(* Version history:
Date	|	Version/Author |	Remark
----------------------------------------------------------------------------------------------------
11.09.01	|	2.01 JP		|	new version depending on 0.99D
22.11.01	|	2.02 JP		|	new version depending on 0.99F
18.01.02	|	2.03 JP		|	new version depending on 1.0
		|				|	changed names, interfaces, execute behavior
25.01.02	|	2.04 JP		|	no CAMMING, change behavior of MC_Power
07.02.02	|	2.05 JP		|	SetOverride in unit less than 1%
13.02.02	|	2.06 JP		|	New: MC_NewPos and MC_NewPosAndVelo
		|				|	removed MC_MoveAdditive
14.02.02	|	2.07 JP		|	completed: MC_Home, MC_MoveSuperImposed
14.02.02	|	2.08 JP		|	renamed MC_NewPosAndVelo New: MC_SetOverride edge triggered
15.02.02	|	2.09 JP		|	changed: MC_Gear
15.02.02	|	2.10 JP		|	changed: MC_SetOverride
04.04.02	|	2.11 JP		|	changed: done for MC_Home 
		|				|	new: Check TimeOut for MoveAbsolute, MoveRelative, Home
08.03.02	|	2.12 JP		|	changed: new flag inserted 
12.03.02	|	2.13 JP		|	changed: reset of bNotExecute
18.03.02	|	2.14 JP		|	changed: MC_Reset waits for ready
22.03.02	|	2.15 JP		|	changed: MC_Read and Write FBs
26.03.02	|	2.16 JP		|	revised: Read/Write Parameter FBs
27.03.02	|	2.17 JP		|	revised: Read/Write Parameter FBs and Home (calibration cam)
09.04.02	|	2.18 JP		|	changed parameter type of some parameters
17.04.02	|	2.19 JP		|	changed: Read(Bool)Parameter new Input to select read mode
							Boolean parameters can be read with ReadParameter
							changed MC_Power: new input override !!			
23.04.02	|	2.20 JP		|	fixed: MC_Home changed: Behavior of MC_MoveAbsolute/Relative
25.04.02	|	2.21 JP		|	changed: MC_Reset: now not waiting for 'axis is ready'. Check with MC_Power !
26.04.02	|	2.22 JP		|	MC_Home: If Posistion =  DEFAULT_HOME_POSITION --> no set of position
							MC_MoveXX: more detailed error messages
05.07.02	|	2.23 JP		|	new MC_MoveAbsoluteOrRestart: combines MoveAbsolute and NewPos
19.07.02	|	2.24 JP		|	changed: E_STATES ---> E_TCMC_STATES
12.09.02	|	2.25 KST		|	changed: MC_MoveAbsolute and MC_MoveRelative now based on FB_MoveGeneric
							MC_NewPos and MC_NewPosAndVelo based on new FB_NewPosAndVeloGeneric 
							new internal start types in MC_MoveAbsoluteOrRestart (message suppression)
16.09.02	|	2.26 ChristophC|	changed: MC_SetActualPosition due to changes in TcNC.Lib
16.10.02	|	2.27 KST		|	new: MC_ExtSetPointGenEnable and MC_ExtSetPointGenDisable
29.10.02	|	2.28 ChristophC|	MC_Stop and MC_SetActualPosition: Ads port changed from TcMcGlobal.NCPORT_TCMC => AMSPORT_R0_NCSAF
12.11.02	|	2.29 ChristophC|	MC_OverrideFilter function block added
13.12.02	|	2.30 JP		|	several smaller changes: MC_ReadStatus, MC_Stop
22.01.03	|	2.31 KSt		|	new additional function MC_ExtSetPointGenFeed
24.03.03	|	2.32 JP		|	added: MC_GearFloat, corr. MC_ReadBoolParameter (wrong for AxisEnPostionRangeMonitoring)
26.03.03	|	2.33 KSt		|	added: MC_MoveModulo
04.04.03	|	2.34 KSt		|	changed: MC_MoveAbsoluteOrRestart, Done will be reset at once after Execute=FALSE
12.05.03	|	2.35 JP		|	changed: MC_MoveVelocity, MC_Home (error handling), MC_ReadStatus
14.05.03	|	2.36 KSt		|	changed: MC_Home, MC_MoveAbsoluteOrRestart
15.05.03	|	2.36.1 KSt	|	changed: MC_Home
28.05.03	|	2.37 KSt		|	changed: MC_MoveVelocity, abort during acceleration phase	
							changed: MC_MoveAbsoluteOrRestart, reset internal error on restart
27.06.03	|	2.38 JP		|	changed: MC_Stop: Execute behavior
22.07.03	|	2.38.1 KSt	|	added: new error codes
12.08.03	|	2.39 KSt		|	changed: FB_ReadWriteParameter, size of bool parameters
15.08.03	|	2.40 KSt		|	added: new block MC_ChangeDynParam
19.08.03	|	2.41 JP		|	changed: MC_ReadParameter: Done falls with Execute
01.10.03	|	2.42 KSt		|	changed: MC_MoveAbsoluteOrRestart, Execute directly after done issue fixed
09.10.03	|	2.43 KSt		|	new function block MC_SetReferenceFlag
04.12.03	|	2.44 KSt		|	ReadBoolParameter(AxisEnTargetPositionMonitoring) corrected
12.01.04	|	2.45 KSt		|	MC_MoveSuperimposed revised
						|	R_Trigger(execute) moved outside CASE in all move function blocks
19.01.04	|	2.45.1 KSt	|	Busy Signal in MC_MoveSuperimposed
30.04.04	|	2.46.0 KSt	|	New function blocks MC_TouchProbe, MC_AbortTrigger, internal block MC_OrientedStop
						|	MC_ReadParameter revised
06.05.04	|	2.46.1 KSt	|	Correction in MC_OrientedStop
21.05.04	|	2.47.0 KSt	|	MC_GearInDyn added - master slave coupling with dynamic gear ratio
06.08.04	|	2.47.1 KSt	|	MC_OrientedStop moved from internal to additional folder
						|	MC_MoveAbsoluteOrRestart additional internal error code NC_ERROR_STARTINTERNAL_NOTREADY evaluated
23.08.04	|	2.47.2 KSt	|	new local flag EmergencyStop in MC_Stop signals type of internal ADS stop command
10.01.05	|	2.47.3 KSt	|	new function block MC_MoveSuperImposedExt
28.01.05	|	2.47.4 KSt	|	TcMcGlobal.tTargetPosTimeOut changed from 5 sec to 6 sec to be later than a NC PEH error (5 sec)
15.02.05	|	2.48.0 KSt	|	new function block MC_GearOutExt 
28.02.05	|	2.49.0 JP		|	Execute and Done behavior corrected for MC_ReadActualPos and MC_SetActualPos
10.03.05	|	2.50.0 KSt	|	all function blocks use a global AMS net-ID TcMcGlobal.NCNETID_TCMC which may be modified by the user
17.03.05	|	2.51.0 KSt	|	new function block MC_PowerStepper
						|	MC_MoveAbsoluteOrRestart restart while starting (adswrite.Busy) changed
24.05.05	|	2.52.0 KSt	|	acceleration added to block MC_GearOutExt 
05.07.05	|	2.53.0 KSt	|	new local flag ADSbusy in all function blocks
05.07.05	|	2.54.0 KSt	|	new function block MC_GearInDynCCV
06.07.05	|	2.55.0 KSt	|	Busy timing improved in all function blocks (turns immediately to FALSE with Done or Error or Aborted)
25.07.05	|	2.55.1 KSt	|	Change for status output behavior 
26.07.05	|	2.55.2 KSt	|	MC_GearOutExt extended through mode 'oriented stop'
03.08.05	|	2.55.3 KSt	|	Commands MC_MoveAbsoluteOrRestart, MC_NewPos and MC_NewPosAndVelo now directed to port AMSPORT_R0_NCSAF
						|	Summary of other commands to SAF: MC_Stop, MC_OrientedStop, MC_TouchProbe, MC_AbortTrigger, MC_SetReferenceFlag, MC_PowerStepper
14.09.05	|	2.56.0 KSt	|	new function block MC_ParameterizedStop
26.09.05	|	2.56.1 KSt	|	Jerk parameter added to MC_ChangeDynParam. Block moved into the internal folder.
07.11.05	|	2.56.2 KSt	|	internal block FB_ReadCharacteristicValues changed to ADSRDWRT
19.12.05	|	2.56.3 KSt	|	new block MC_SetActualPositionOnTheFly
05.01.06	|	2.56.4 KSt	|	new blocks MC_ReadParameterSet and MC_ReadAxisComponents
21.02.06	|	2.57.0 KSt	|	NC status feedback monitoring changed in MC_GearIn and MC_GearInFloat
29.03.06	|	2.57.1 KSt	|	new order of the blocks in the library tree
11.04.06	|	2.57.2 HKP	|	Command MC_ChangeDynParam now directed to port AMSPORT_R0_NCSAF
10.05.06	|	2.57.3 KSt	|	new function block MC_Jog
17.05.06	|	2.57.4 KSt	|	MC_Jog: MC_JOGMODE_INCHING_MODULO temporarily deactivated
05.07.06	|	2.57.5 KSt	|	NC status feedback monitoring changed in MC_GearInDyn and MC_GearInDynCCV
=======	|===============	|==========================================================================
12.07.06	|	2.57.6 KSt	|	new AMS port NCPORT_TCMC_COUPLING for all coupling commands
11.08.06	|	2.57.7 KSt	|	reset Done when Execute is FALSE in FB_NewPosAndVeloGeneric
						|	MC_Jog released
22.08.06	|	2.57.8 KSt	|	new function block MC_AbortSuperposition
07.11.06	|	2.57.9 HKP	|	changes in function block MC_PowerStepper
06.02.07	|	2.57.10 KSt	|	initialization problem with modulo positions fixed in MC_TouchProbe.
						|	recorded position at PlcEvent now modulo when requested.
14.03.07	|	2.57.11 KSt	|	MC_Jog: Handling of CommandAborted corrected
24.04.07	|	2.57.12 KSt	|	additional parameters in MC_AxisPara, MC_ReadParameters, MC_WriteParameters
31.05.07	|	2.57.13 KSt	|	FPU exception with LREAL_TO_BOOL and DWORD_TO_BOOL fixed in FB_ReadWriteParameter 
12.06.07	|	2.57.14 KSt	|	FB_NewPosAndVeloGeneric and MC_MoveSuperImposed(Ext): IF condition changed from "NOT AxisIsMoving" to "NOT AxisHasJob"
=======	|===============	|==========================================================================
12.06.07	|	2.57.14 KSt	|	TcMC2 development started - following 2.xx.xx changes have been added in parallel
02.11.07	|	2.57.15 KSt	|	data structure ST_TableCharacValues extended
18.12.07	|	2.57.16 KSt	|	MC_Jog is now internally using MC_MoveRelative instead of MC_MoveAbsolute to work with backlash compensation
20.05.08	|	2.57.18 KSt	|	AxisModuloPositionFlag added to MC_ReadBoolParameter
17.06.08	|	2.57.20 KSt	|	MC_GearInMultiMaster added
24.07.08	|	2.57.22 KSt	|	MC_Power supports now a minimum Enable-Off/On toggle time of 50ms to reenable the Status output
28.10.08	|	2.57.23 KSt	|	new function block MC_SetEncoderScalingFactor
=======	|===============	|==========================================================================
16.03.07	|	3.00.00 KSt	|	new version depending on PLCopen V1.1 (beta)
25.08.08   |	3.00.01 KSt	|	released as TcMC2 
17.09.08   |	3.00.02 KSt	|	last result added in MC_Reset
26.11.08   |	3.00.03 KSt	|	change in MC_Stop and MoveGeneric for delayed error handling
01.12.08   |	3.00.04 KSt	|	MC_Stop - Done is set immediately at standstill
18.12.08   |	3.00.05 KSt	|	MC_Power - uses now ControlLoopClosed instead of AxisIsReady
13.01.09   |	3.00.06 KSt	|	independent characteristic data for camming and flying saw
16.01.09   |	3.00.07 KSt	|	all move commands: changed handling of CmdNo=0 and CmdNo+2 leads to better results (CommandAborted)
23.01.09   |	3.00.08 KSt	|	MC_MoveSuperimposed is now passed to port AMSPORT_R0_NCSAF (501)
28.01.09   |	3.00.09 KSt	|	Homing mode MC_Direct added - Mode option for MC_SetPosition added
29.01.09   |	3.00.10 KSt	|	Warning output added to MC_MoveSuperimposed
05.02.09   |	3.00.11 KSt	|	axis state is now DISABLED if control loop is not closed (was STANDSTILL for virtual axes - _F_AxisState)
05.02.09   |	3.00.11 KSt	|	all move commands: CmdNo=0 is ignored as invalid - change of the coupled state leads to CommandAborted
06.02.09   |	3.00.11 KSt	|	errors on missing cyclic NC command feedback are delayed for a few cycles to avoid problems with multiple function block calls during one PLC cycle
19.02.09   |	3.00.12 KSt	|	MC_GearInDyn and MC_GearInMultimaster - no reset of gear ratio after Enable is reset to FALSE
24.02.09   |	3.01.00 KSt	|	Motion commands on slaves (must be enabled in the axis parameters before)
12.03.09   |	3.01.01 KSt	|	MC_Jog - Active output added - reset outputs when Execute is false 
09.04.09   |	3.01.02 KSt	|	MC_SetPosition and MC_SetEncoderScalingFactor - explicit encoder / control loop index 0..n can be selected
15.04.09   |	3.01.03 KSt	|	MC_Stop - outputs (except Busy) are reset after Execute=FALSE - can be retriggered during release phase
17.04.09   |	3.01.04 KSt	|	MC_Home - static homing with DEFAULT_HOME_POSITION implemented - Option.ClearPositionLag available 
11.05.09   |	3.01.05 KSt	|	MC_Stop - incorrect error message 4B63 removed;  
30.06.09   |	3.01.06 KSt	|	MC_MoveSuperimposed - new types ACCREDUCTION - new AbortOptions
28.07.09   |	3.01.07 KSt	|	MC_ExtSetPointGenFeed feeds additional counter information to the NC
13.08.09   |	3.01.08 KSt	|	MC_MoveSuperimposed - new AbortOptions - Done behavior adapted
01.09.09   |	3.01.09 KSt	|	MC_SetPosition - new option 'set absolute measuring'
30.09.09   |	3.01.10 KSt	|	MC_MoveSuperimposed - fix for new AbortOptions - HasJob flag not required before starting the command
06.10.09   |	3.01.11 KSt	|	MC_Stop - wait extra cycles before axis release error 
06.10.09   |	3.01.12 KSt	|	MC_MoveSuperimposed - fix for new AbortOptions - HasJob or IsMoving check at beginning and end of compensation 
07.10.09   |	3.01.13 KSt	|	MC_MoveSuperimposed - initial motion check removed for new AbortOptions
28.10.09   |	3.01.14 KSt	|	MC_ExtSetPointGenEnable/Disable - port changed from SVB to SAF
06.11.09   |	3.01.15 KSt	|	MC_SetPosition - new option 'set absolute measuring' removed
09.11.09   |	3.01.16 KSt	|	MC_Stop on slave axes was not rejected with error - fixed
18.11.09   |	3.01.17 KSt	|	MC_Jog - usage with protected (coupled) axes refused
26.11.09   |	3.01.18 KSt	|	Axis status data: UpdateCycleTime calculation fixed
08.12.09   |	3.01.19 KSt	|	_FB_MoveGeneric - mapping check to avoid early Error and CommandAborted signals
25.02.10   |	3.01.20 KSt	|	MC_MoveSuperimposed - additional outputs ActualAcceleration and ActualDeceleration
11.03.10   |	3.01.21 KSt	|	MC_Power - no Enable timeout error for coupled axes
07.04.10   |	3.01.22 KSt	|	MC_ReadApplicationRequest added
15.04.10   |	3.01.23 KSt	|	MC_PositionCorrectionLimiter added - cyclic update of UpdateTaskIndex and UpdateCycleTime removed from ReadStatus
23.04.10   |	3.01.24 KSt	|	internal MC_TouchProbe_V2_00 for new multi probe interface
04.05.10   |	3.01.25 KSt	|	fix in MC_WriteParameter to write bool parameters with MC_WriteParameter as well as MC_WriteBoolParameters
06.05.10   |	3.01.25 KSt	|	fix in MC_MoveContinous... for output InEndVelocity
31.05.10   |	3.02.00 KSt	|	_TcMC_ADS commands added to allow PLC running faster than NC, added to MC_Reset
08.07.10   |	3.02.01 KSt	|	fix in NC mapping counter monitoring (time-out check)
24.09.10   |	3.02.02 KSt	|	ST_NcApplicationRequest structure extended
27.10.10   |	3.02.03 KSt	|	MC_TouchProbe - TRUNC function replaced by MODABS for modulo calculations
22.11.10	|	3.02.04 KSt	|	MC_Power - axis will be enabled automatically after Error turns to FALSE and control loop is closed (just if Enable=TRUE)
		|				|	Move-Commands on axes with external set point generator (must be enabled in the axis parameters before)
29.11.10	|	3.02.05 KSt	|	MC_ReadParameter - new parameters AxisCycleTime NcSafCycleTime and NcSvbCycleTime
17.01.11	|	3.02.06 KSt	|	Phasing blocks added
21.01.11	|	3.02.06 KSt	|	MC_ExtSetPointGenEnable and MC_ExtSetPointGenDisable: code rewritten in ST
16.02.11	|	3.02.07 KSt	|	MC_TouchProbe and MC_TouchProbe_V2_00 - correction for WindowOnly with FirstPosition>LastPosition
18.02.11	|	3.02.08 KSt	|	MC_TouchProbe_V2_00 - TRIGGER_REF extended by optional physical input definition 
21.02.11	|	3.02.08 KSt	|	_MC_Phasing beta version included
25.03.11	|	3.02.09 KSt	|	minor adaption to PlcOpen V2.0 "Function blocks for motion control" released document.
05.04.11	|	3.02.10 KSt	|	new parameters defined for fast axis stopp 
21.04.11	|	3.02.11 KSt	|	FB_MoveUniversalGeneric - fix in command number overrun calculation 
27.04.11	|	3.02.12 KSt	|	new function block MC_ReadStopInfo to read the expected distance and time to stop an axis
02.05.11	|	3.02.13 KSt	|	dynamical data for fast axis stopp can be read or written by MC_ReadParameter, MC_WriteParameter
03.05.11	|	3.02.14 KSt	|	MC_TouchProbe_V2_00 - additional output data structure MC_TouchProbeRecordedData 
11.05.11	|	3.02.15 KSt	|	type check adaptions for the PLC3 compiler
18.05.11	|	3.02.16 KSt	|	data types ST_AxisParameterSet and ST_NcApplicationRequest extended
31.05.11	|	3.02.17 HKP	|	Check of AxisIsReady removed from MC_MoveCommands
31.05.11	|	3.02.17 KSt	|	Axis.OpMode.SimulationAxis added
29.06.11	|	3.02.18 KSt	|	MC_ReadParameterSet fixed for use with differently aligned systems (ARM)
12.07.11	|	3.02.19 KSt	|	internal storage added to AXIS_REF
19.07.11	|	3.02.20 KSt	|	Two Speed Axes: InVelocity detection fixed in MC_MoveVelocity
01.08.11	|	3.02.21 KSt	|	Check of cyclic motion command call - 'buffered command monitoring error' changed to 'cyclic call error' if not cyclically called
07.09.11	|	3.02.22 KSt	|	optional advanced slave motion profile for MC_GearInMultiMaster
13.10.11	|	3.02.23 KSt	|	new OpMode flag AllowExtSetAxisCommands
08.12.11	|	3.02.25 KSt	|	stop monitoring for stop and halt commands added (comparable with target position monitoring)
22.12.11	|	3.02.26 KSt	|	MC_Reset fixed for short PLC cycle times (_TcMC_ADSWRITE waits 2 cycles for NC process image)
22.12.11	|	3.02.27 KSt	|	MC_GearOut and MC_CamOut are now waiting for the NC couple state feedback in Nc2Plc
19.01.12	|	3.02.28 KSt	|	MC_TouchProbe_V2 released
23.02.12	|	3.02.29 ICh	|	_ST_TcNc_OperationModes: cleanup, StopMonitoring added, _ST_TcNC_SetPos: fReserved added to match NC definition
23.02.12	|	3.02.30 KSt	|	typecasts for TC3 to avoid TC3 compiler messages
23.03.12	|	3.02.31 KSt	|	initialization code for MoveModulo revised 
16.05.12	|	3.02.32 KSt	|	MC_MoveVelocity: InVelocity is now reset after abortion or error
05.07.12	|	3.02.33 KSt	|	state diagram changed - if axis has error, state is always ERRORSTOP (never DISABLED)
27.07.12	|	3.02.34 KSt	|	new function blocks MC_BacklashCompensation and MC_TableBasedPositionCompensation. MC_PositionCorrectionLimiter: Acceleration=0 means disables limitation.
23.08.12	|	3.02.35 KSt	|	MC_Power now avoids time out errors after an axis reset
04.04.13	|	3.02.36 KSt	|	extended ST_DriveAddress structure; used with MC_ReadDriveAddress
02.07.13	|	3.02.37 KSt	|	Done may have come together with Error or CommandAborted - fixed by resetting Done in these cases.
10.07.13	|	3.02.38 KSt	|	MC_Move commands now check NC interface update before monitoring NC feedback
02.09.13	|	3.02.39 KSt	|	MC_PositionCorrectionLimiter - mode UNLIMITED for axes in standstill fixed (was internally set to FAST before)
04.09.13	|	3.02.40 KSt	|	now waiting for READDEVINFO (NC version) in MC_AbortTrigger_V2_00 and MC_ReadDriveAddress
01.10.13	|	3.02.41 KSt	|	function MC_SetAcceptBlockedDriveSignal added
01.10.13	|	3.02.42 KSt	|	debug message for positive move commands can be enabled with ControlDWord.29
22.11.13	|	3.02.43 KSt	|	Avoid too early Active output at Move commands - now waiting for NcToPlc mapping after ADS command
21.03.14	|	3.02.44 KSt	|	MC_AbortTrigger now falls back to initialization state and resets busy after operration
20.05.14	|	3.02.45 KSt	|	correction of Status.UpdateCycleTime in _F_ReadStatus
14.07.14	|	3.02.46 KSt	|	MC_ReadParameter, MC_WriteParameter, Port changed to 501 for parameters AxisRemainingTimeToGo and AxisRemainingDistanceToGo
22.10.14	|	3.02.47 KSt	|	MC_Move commands Active feedback optimized. Active now turns to true as soon as the CmdNo has definitely changed and is equal to own number (NC response).
23.10.14	|	3.02.48 KSt	|	MC_BacklashCompensation - Correction in parameter check
30.09.14	|	3.02.49 KSt	|	MC_MoveSuperimposed and MC_AbortSuperposition now redirected to NCPORT_TCMC_SUPERPOSITION, port can be modified by user
19.03.15	|	3.02.50 KSt	|	MC_Stop command can now be aborted by a reset command if axis is in standstill and the flag "Motion Commands Locked" is false
05.05.15	|	3.02.51 KSt	|	MC_Power - error feedback in case of axis errors corrected 
03.08.15	|	3.02.51b KSt|	TC3 only, new blocks MC_WriteParameterPersistent and MC_WriteBoolParameterPersistent
25.09.15	|	3.02.51c Fap|	TC3 only, additional internal InGear2 flag for MC_GearInMultiMaster
*)


CASE nVersionElement OF
1:	(* major number *)
	F_GetVersion_TcMC2 := 3;
2:	(* minor number *)
	F_GetVersion_TcMC2 := 3;
3:	(* revision number *)
	F_GetVersion_TcMC2 := 38;
ELSE
	F_GetVersion_TcMC2 := 16#FFFF;
END_CASE

END_FUNCTION

// POUs/Administrative/Axis Functions/MC_Power
{attribute 'conditionalshow_all_locals'}
FUNCTION_BLOCK MC_Power
(*
	Function block defined by PLCopen Part 1 - Function blocks for motion control

	This Function Block controls the power stage (on or off).

	Only 1 FB MC_Power should be issued per axis.
*)
VAR_IN_OUT
	Axis				:	AXIS_REF; (*Reference to an axis*)
END_VAR
VAR_INPUT
	Enable			:	BOOL;	(* B *)
	Enable_Positive	:	BOOL;	(* E *)
	Enable_Negative	:	BOOL;	(* E *)
	Override		:	LREAL	(* V *) 	:= 100.0; (* in percent - Beckhoff proprietary input *)
	BufferMode		:	MC_BufferMode;	(* V *)	
	Options			:	ST_PowerOptions;
END_VAR
VAR_OUTPUT
	Status			:	BOOL;	(* B *)
	Busy			: 	BOOL;	(* V *)
	Active			: 	BOOL;	(* V *)
(*	Valid			: 	BOOL;*)	(* E *)	(* not implemented - use Busy *)
	Error			:	BOOL;	(* B *)
{attribute 'displaymode':='hex'}
	ErrorID			:	UDINT;	(* E *)
END_VAR
VAR
	EnableTimeout: TON;
	EnableOffOnDelay: TP;
(*	iOverride: DINT;*)
	iOverride: DWORD;	(* 20110511 KSt type adaption for TC3 *)
END_VAR

IF NOT _F_TcMC_IsValidAxisRef(Axis) THEN // AXIS REFERENCE CHECK - 2020-09-17 KSt
	Error := TRUE;
	ErrorID := MC_ERROR_INVALIDREFERENCE;
	RETURN;
END_IF

(*
	PlcOpen comment zu MC_Power:
		Eingänge >Override< und >BufferMode< sind Beckhoff-spezifisch 
		Ausgänge >Busy< und >Active< sind Beckhoff-spezifisch 
		Ausgang >Valid< fehlt, Funktion entspricht Active 
*)

(*EnableTimeout(IN:=Enable, PT:=T#10s);*)	(* timout if axis doesn't get ready after Enable *)
(*EnableTimeout(IN:=Enable AND NOT Status AND Axis.NcToPlc.CoupleState=0, PT:=T#10s);*) (* 2012-08-23 KSt *)	(* timout if axis doesn't get ready after Enable - just for single axes - KSt 2010-03-11 *)
(*EnableTimeout(IN:=Enable AND NOT Status AND Axis.NcToPlc.CoupleState=0 AND Axis.NcToPlc.ErrorCode=0, PT:=T#10s);*)(* 2012-08-23 KSt *) (* timout if axis doesn't get ready after Enable - just for single axes and only if error free - KSt 2012-08-23 *)
EnableTimeout(IN:=Enable AND NOT Status AND Axis.NcToPlc.CoupleState=0 AND Axis.NcToPlc.ErrorCode=0, PT:=T#16S);	(* 2021-02-01 KSt *) (* timeout changed from 10 to 16 s since NC reaction may take up to 15 s in case of drive reset issues *)
EnableOffOnDelay(IN:= NOT Enable );	(* minimum delay between disable end re-Enable -  don't initialize before first enable *)

IF Enable THEN
	Busy := TRUE;
	Status := FALSE;
	ErrorID := 0;
	Error := FALSE;
	EnableOffOnDelay.PT:=T#50ms;	(* initialize not before first enable *)

	(* set override *)
	iOverride := LREAL_TO_DWORD(Override*10000);
	(* double check override with real and integer number because conversion may fail *)
	IF (Override < -1) OR (Override > 101) THEN	(* check real number with tolerance *)
		ErrorID := MC_ERROR_PARAMETER_NOT_CORRECT;
		Error := TRUE;
	ELSIF (iOverride < 0) OR (iOverride > 1000000) THEN	(* check integer number without tolerance *)
		ErrorID := MC_ERROR_PARAMETER_NOT_CORRECT;
		Error := TRUE;
	ELSE
		Axis.PlcToNc.Override := iOverride;
	END_IF;

	(* set enabling flags *)
	Axis.PlcToNc.ControlDWord.0 := Enable;
	Axis.PlcToNc.ControlDWord.1 := Enable_Positive;
	Axis.PlcToNc.ControlDWord.2 := Enable_Negative;

	(* set status bit *)
	(* IF  F_AxisIsReady(StateDWord := Axis.NcToPlc.StateDWord) THEN *) (* Axis ready*) 	(* 2008-12-18 KSt *)
	IF  F_AxisControlLoopClosed(StateDWord := Axis.NcToPlc.StateDWord) THEN (* Axis ready*) 	(* 2008-12-18 KSt *)
		(* status is TRUE if no error and a minimum of EnableOffOnDelay.PT (50 ms) after last recent disable *)
(*		Status := NOT Error AND NOT EnableOffOnDelay.Q; *)(* exclusive outputs *)

		(* 20101122 KSt - If control loop is closed after an error, the error is reset and the axis status is enabled *)
		(* status is TRUE after a minimum EnableOffOnDelay.PT (50 ms) after last recent disable *)
		Status := NOT EnableOffOnDelay.Q;
		IF Status THEN (* exclusive outputs *)
			Error := FALSE;
			ErrorID := 0;
		END_IF
	(*	ELSIF Axis.Status.ErrorID <> 0 THEN *)(* 2009-01-29 KSt *)
	ELSIF Axis.NcToPlc.ErrorCode <> 0 THEN (* 2012-08-23 KSt *)
		Status := FALSE;
		Error := TRUE;
		(* ErrorID := Axis.Status.ErrorID;*)	(* 2015-05-05 KSt *)
		ErrorID := Axis.NcToPlc.ErrorCode;	(* 2015-05-05 KSt *)
	ELSIF EnableTimeout.Q THEN
		(* timeout after enable *)
		Status := FALSE;
		Error := TRUE;
		ErrorID := MC_ERROR_AXIS_IS_NOT_READY;
	END_IF;

ELSE (* NOT Enable *)
	(* if BufferMode=Buffered wait for current command beeing finished *)
	IF BufferMode = MC_Aborting OR NOT F_AxisHasJob(Axis.NcToPlc.StateDWord) THEN
(* changed 20100416 KSt *) (*
		Axis.PlcToNc.ControlDWord:= CLEARBIT32(Axis.PlcToNc.ControlDWord,0);
		Axis.PlcToNc.ControlDWord:= CLEARBIT32(Axis.PlcToNc.ControlDWord,1);
		Axis.PlcToNc.ControlDWord:= CLEARBIT32(Axis.PlcToNc.ControlDWord,2);	*)
		Axis.PlcToNc.ControlDWord.0 := FALSE;
		Axis.PlcToNc.ControlDWord.1 := FALSE;
		Axis.PlcToNc.ControlDWord.2:= FALSE;
		(* Override  0 % *)
		Axis.PlcToNc.Override := 0;
		Status := FALSE;
		Busy := FALSE;
		Error := FALSE;			(* reset at falling edge of Execute *)
		ErrorID := 0;
	END_IF
END_IF;

Active:=TRUE;

END_FUNCTION_BLOCK

// POUs/Motion/Point To Point Motion/MC_MoveAdditive
FUNCTION_BLOCK MC_MoveAdditive
(*	This Function Block commands a controlled motion of a specified relative
	distance additional to the most recent commanded position in the discrete 
	motion state. The most recent commanded position may be the result of a 
	previous MC_MoveAdditive motion which was aborted. If the FB is activated 
	in the Continuous Mode the specified relative distance is added to the actual 
	position at the time of the execution.

 	MC_MoveAdditive ist ähnlich MC_MoveRelative. Wenn während der Bewegung
	getriggert, dann wird allerdings die ursprüngliche Zielposition um Distance 
	verlängert. Eine Endlosachse wird in eine diskrete Bewegung ausgehend 
	von der aktuellen Position plus Distanz gewandelt.
*)
VAR_IN_OUT
	Axis				:	AXIS_REF; (*Reference to an axis*)
END_VAR
VAR_INPUT
	Execute			:	BOOL;	
(*	ContinuousUpdate :	BOOL; *)		(* not available *)
	Distance			:	LREAL;	
	Velocity			:	LREAL;	
	Acceleration		:	LREAL;	
	Deceleration		:	LREAL;	
	Jerk				:	LREAL;	
	BufferMode		:	MC_BufferMode;	
	Options			: 	ST_MoveOptions;	
END_VAR
VAR_OUTPUT
	Done			:	BOOL;	
	Busy			: 	BOOL;	
	Active			: 	BOOL;	
	CommandAborted	:	BOOL;	
	Error			:	BOOL;	
{attribute 'displaymode':='hex'}
	ErrorID			:	UDINT;	
END_VAR
VAR
	LastExecutionResult: 	_ST_FunctionBlockResults;
	ADSbusy		: 	BOOL;
	MoveGeneric		: 	_FB_MoveUniversalGeneric;
	CmdNo: UINT;
END_VAR

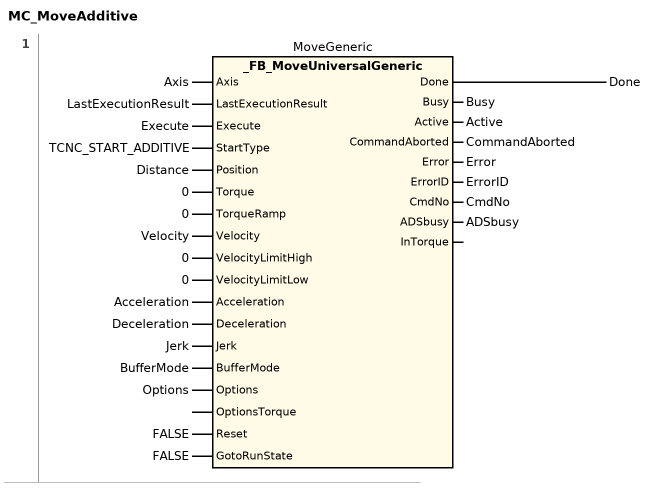
// NETWORK 1
MoveGeneric(
    Axis := Axis,
    LastExecutionResult := LastExecutionResult,
    Execute := Execute,
    StartType := TCNC_START_ADDITIVE,
    Position := Distance,
    Torque := 0,
    TorqueRamp := 0,
    Velocity := Velocity,
    VelocityLimitHigh := 0,
    VelocityLimitLow := 0,
    Acceleration := Acceleration,
    Deceleration := Deceleration,
    Jerk := Jerk,
    BufferMode := BufferMode,
    Options := Options,
    Reset := FALSE,
    GotoRunState := FALSE,
    Busy => Busy,
    Active => Active,
    CommandAborted => CommandAborted,
    Error => Error,
    ErrorID => ErrorID,
    CmdNo => CmdNo,
    ADSbusy => ADSbusy); // _FB_MoveUniversalGeneric
Done := MoveGeneric.Done;

END_FUNCTION_BLOCK

// POUs/Motion/Point To Point Motion/MC_MoveRelative
FUNCTION_BLOCK MC_MoveRelative
(*	This Function Block commands a controlled motion of a specified distance
	relative to the actual position at the time of the execution.
*)
VAR_IN_OUT
	Axis				:	AXIS_REF; (*Reference to an axis*)
END_VAR
VAR_INPUT
	Execute			:	BOOL;	
(*	ContinuousUpdate :	BOOL; *)		(* not available *)
	Distance			:	LREAL;	
	Velocity			:	LREAL;	
	Acceleration		:	LREAL;	
	Deceleration		:	LREAL;	
	Jerk				:	LREAL;	
	BufferMode		:	MC_BufferMode;	
	Options			: 	ST_MoveOptions;	
END_VAR
VAR_OUTPUT
	Done			:	BOOL;	
	Busy			: 	BOOL;	
	Active			: 	BOOL;	
	CommandAborted	:	BOOL;	
	Error			:	BOOL;	
{attribute 'displaymode':='hex'}
	ErrorID			:	UDINT;	
END_VAR
VAR
	LastExecutionResult: 	_ST_FunctionBlockResults;
	ADSbusy		: 	BOOL;
	MoveGeneric		: 	_FB_MoveUniversalGeneric;
	CmdNo: UINT;
END_VAR

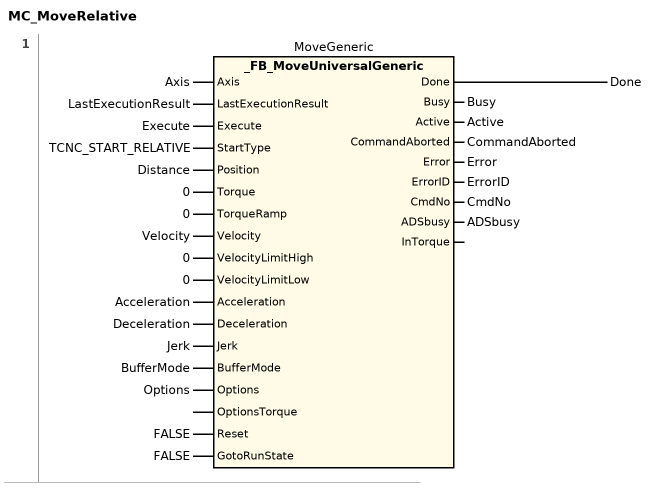
// NETWORK 1
MoveGeneric(
    Axis := Axis,
    LastExecutionResult := LastExecutionResult,
    Execute := Execute,
    StartType := TCNC_START_RELATIVE,
    Position := Distance,
    Torque := 0,
    TorqueRamp := 0,
    Velocity := Velocity,
    VelocityLimitHigh := 0,
    VelocityLimitLow := 0,
    Acceleration := Acceleration,
    Deceleration := Deceleration,
    Jerk := Jerk,
    BufferMode := BufferMode,
    Options := Options,
    Reset := FALSE,
    GotoRunState := FALSE,
    Busy => Busy,
    Active => Active,
    CommandAborted => CommandAborted,
    Error => Error,
    ErrorID => ErrorID,
    CmdNo => CmdNo,
    ADSbusy => ADSbusy); // _FB_MoveUniversalGeneric
Done := MoveGeneric.Done;

END_FUNCTION_BLOCK

// POUs/Motion/Homing/MC_Home
{attribute 'conditionalshow_all_locals'}
FUNCTION_BLOCK MC_Home
(*
	Function block defined by PLCopen Part 1 - Function blocks for motion control

	This Function Block commands the axis to perform the «search home» sequence.
	The details of this sequence can be set by the axis parameters. 
	The 'Position' input is used to set the absolute position when reference signal 
	is detected. This Function Bock completes at 'StandStill'.
*)
VAR_IN_OUT
	Axis				:	AXIS_REF; (*Reference to an axis*)
END_VAR
VAR_INPUT
	Execute				:	BOOL;	
	Position			:	LREAL	 := DEFAULT_HOME_POSITION;
	HomingMode			: 	MC_HomingMode;	
	BufferMode			:	MC_BufferMode;	
	Options				: 	ST_HomingOptions;		(* Beckhoff proprietary input *)
	bCalibrationCam 	: 	BOOL;		(* Beckhoff proprietary input *)
END_VAR
VAR_OUTPUT
	Done				:	BOOL;	
	Busy				: 	BOOL;	
	Active				: 	BOOL;	
	CommandAborted		:	BOOL;	
	Error				:	BOOL;	
{attribute 'displaymode':='hex'}
	ErrorID				:	UDINT;	
END_VAR
VAR
	LastExecutionResult	: 	_ST_FunctionBlockResults;
	ADSbusy				: 	BOOL;
	iState				: 	_E_TcMC_STATES := STATE_INITIALIZATION;
	iSubState			: 	INT;
	fbAdsWriteCmd		: 	ADSWRITE;
	fbAdsWriteParameter	: 	ADSWRITE; // 2018-02-05 FAP added homing parameters to options
	fbAdsReadRefPos		: 	ADSREAD;
	ReferenceFlagValue	: UDINT;
	fbSetPosition		: MC_SetPosition;

	CalibrationValue	: LREAL;
	SearchDirection		: UINT;
	SearchVelocity		: LREAL;
	SyncDirection		: UINT;
	SyncVelocity		: LREAL;
	ReferenceMode		: E_EncoderReferenceMode;
END_VAR
VAR
{attribute 'conditionalshow'}
	fbTrigger			:	R_TRIG;
{attribute 'conditionalshow'}
	fbTimeOut			:	TON;
END_VAR


(*
	PlcOpen comment to MC_Home:
		HomingMode input ist Beckhoff-spezifisch (war in vorheriger Spezifikation mal vorhanden)
		BufferMode ist nicht implementiert.
*)

 fbTrigger(CLK:= Execute);

CASE iSubState OF
	0 :	(* init *)
		iState := STATE_INITIALIZATION;	(* *)
		Busy := FALSE;
		IF NOT Execute THEN
			Done := FALSE;
			CommandAborted := FALSE;
			Error := FALSE;			(* reset at falling edge of Execute *)
			ErrorID := 0;
		END_IF
	   	IF fbTrigger.Q THEN
			(* initialize output values *)
	   		Busy := TRUE;
			Done := FALSE;
			CommandAborted := FALSE;
			Error := FALSE;
			ErrorID := 0;
			fbAdsWriteCmd(WRITE:=FALSE);
//			fbAdsWriteRefPos(WRITE:=FALSE); 2018-02-05 FAP added homing parameters to options
			fbAdsWriteParameter(WRITE:=FALSE);
			fbAdsReadRefPos(READ:=FALSE);
			fbTimeOut(IN:=FALSE);
			fbSetPosition(	Execute:= FALSE, Axis:=Axis);

			IF BufferMode <> 0 THEN
		   		Busy := FALSE;
				Error := TRUE;
				ErrorID := MC_ERROR_BUFFERMODE_NOT_SUPPORTED;
			ELSIF (Options.SearchDirection <> MC_Direction.MC_Positive_Direction 
					AND Options.SearchDirection <> MC_Direction.MC_Negative_Direction 
					AND Options.SearchDirection <> MC_Direction.MC_Undefined_Direction)
			  OR (Options.SyncDirection <> MC_Direction.MC_Positive_Direction
			  		AND Options.SyncDirection <> MC_Direction.MC_Negative_Direction
			  		AND Options.SyncDirection <> MC_Direction.MC_Undefined_Direction)
			  OR Options.SearchVelocity < 0.0
			  OR Options.SyncVelocity < 0.0
			  OR Options.ReferenceMode > ENCODERREFERENCEMODE_SOFTDRIVELATCHNEG 
			  OR Options.ReferenceMode < ENCODERREFERENCEMODE_DEFAULT THEN
		   		Busy := FALSE;
				Error := TRUE;
				ErrorID := MC_ERROR_PARAMETER_NOT_CORRECT;				
			ELSE
				CASE HomingMode OF
					MC_DefaultHoming :
						IF Position < DEFAULT_HOME_POSITION THEN
							iSubState := iSubState + 1;	(* Write homing calibration value *)
						ELSIF Options.SearchDirection <> MC_Direction.MC_Undefined_Direction THEN
							iSubState := iSubState + 2;	(* Write homing search direction *)
						ELSIF Options.SearchVelocity > 0.0 THEN
							iSubState := iSubState + 3;	(* Write homing search velocity *)
						ELSIF Options.SyncDirection <> MC_Direction.MC_Undefined_Direction THEN
							iSubState := iSubState + 4;	(* Write homing sync direction *)
						ELSIF Options.SyncVelocity > 0.0 THEN
							iSubState := iSubState + 5;	(* Write homing sync velocity *)
						ELSIF Options.ReferenceMode <> E_EncoderReferenceMode.ENCODERREFERENCEMODE_DEFAULT THEN
							iSubState := iSubState + 6;	(* Write homing reference mode *)
						ELSE
							iSubState := 11; 	(* start homing (isubState = 11) *)
						END_IF
					MC_Direct :
						ReferenceFlagValue := 1;
						IF Position < DEFAULT_HOME_POSITION THEN
							fbSetPosition.Position := Position;
							iSubState := 22;	(* set position and reference flag *)
						ELSE
							iSubState := 21; 	(* read homing position and then set position and reference flag *)
						END_IF
					MC_ForceCalibration :
						ReferenceFlagValue := 1;
						iSubState := 31; (* set reference flag *)
					MC_ResetCalibration :
						ReferenceFlagValue := 0;
						iSubState := 31; (* set reference flag *)
				ELSE (* case *)
			   		Busy := FALSE;
					Error := TRUE;
					ErrorID := MC_ERROR_CALIBRATION_ERROR; (* homing mode not supported *)
				END_CASE
			END_IF
		END_IF

	1: // Write homing calibration value
		CalibrationValue := Position;
		fbAdsWriteParameter(	NETID:= TcMcGlobal.NCNETID_TCMC,
								PORT:= TcMcGlobal.NCPORT_TCMC,
								IDXGRP:=TcMcGlobal.Axis.Parameter.IDXGRP+Axis.NcToPlc.AxisId,
								IDXOFFS:= TcMcGlobal.Axis.Parameter.IDXOFFS.REF_POS,
								LEN:= SIZEOF(CalibrationValue),
								SRCADDR:= ADR(CalibrationValue),
								WRITE:= TRUE,
								TMOUT:= TcMcGlobal.tADSTimeOut);
		IF NOT fbAdsWriteParameter.Busy THEN
			IF fbAdsWriteParameter.Err	THEN
				Error := fbAdsWriteParameter.ERR;
				ErrorID := fbAdsWriteParameter.ERRID;
				iSubState := 0;
			ELSE
				IF Options.SearchDirection <> MC_Direction.MC_Undefined_Direction THEN
					iSubState := iSubState + 1;	(* Write homing search direction *)
				ELSIF Options.SearchVelocity > 0.0 THEN
					iSubState := iSubState + 2;	(* Write homing search velocity *)
				ELSIF Options.SyncDirection <> MC_Direction.MC_Undefined_Direction THEN
					iSubState := iSubState + 3;	(* Write homing sync direction *)
				ELSIF Options.SyncVelocity > 0.0 THEN
					iSubState := iSubState + 4;	(* Write homing sync velocity *)
				ELSIF Options.ReferenceMode <> E_EncoderReferenceMode.ENCODERREFERENCEMODE_DEFAULT THEN
					iSubState := iSubState + 5;	(* Write homing reference mode *)
				ELSE
					iSubState := 11; 	(* start homing (isubState = 11) *)
				END_IF
			END_IF
			fbAdsWriteParameter(WRITE:=FALSE);
		END_IF

	2: // Write homing search direction
		SearchDirection := SEL(Options.SearchDirection = MC_Direction.MC_Positive_Direction, 1, 0);
		fbAdsWriteParameter(	NETID:= TcMcGlobal.NCNETID_TCMC,
								PORT:= TcMcGlobal.NCPORT_TCMC,
								IDXGRP:=TcMcGlobal.Axis.Parameter.IDXGRP+Axis.NcToPlc.AxisId,
								IDXOFFS:= TcMcGlobal.Axis.Parameter.IDXOFFS.ENCSEARCHDIR,
								LEN:= SIZEOF(SearchDirection),
								SRCADDR:= ADR(SearchDirection),
								WRITE:= TRUE,
								TMOUT:= TcMcGlobal.tADSTimeOut);
		IF NOT fbAdsWriteParameter.Busy THEN
			IF fbAdsWriteParameter.Err	THEN
				Error := fbAdsWriteParameter.ERR;
				ErrorID := fbAdsWriteParameter.ERRID;
				iSubState := 0;
			ELSE
				IF Options.SearchVelocity > 0.0 THEN
					iSubState := iSubState + 1;	(* Write homing search velocity *)
				ELSIF Options.SyncDirection <> MC_Direction.MC_Undefined_Direction THEN
					iSubState := iSubState + 2;	(* Write homing sync direction *)
				ELSIF Options.SyncVelocity > 0.0 THEN
					iSubState := iSubState + 3;	(* Write homing sync velocity *)
				ELSIF Options.ReferenceMode <> E_EncoderReferenceMode.ENCODERREFERENCEMODE_DEFAULT THEN
					iSubState := iSubState + 4;	(* Write homing reference mode *)
				ELSE
					iSubState := 11; 	(* start homing (isubState = 11) *)
				END_IF
			END_IF
			fbAdsWriteParameter(WRITE:=FALSE);
		END_IF
	
	3: // Write homing search velocity
		SearchVelocity	:= Options.SearchVelocity;
		fbAdsWriteParameter(	NETID:= TcMcGlobal.NCNETID_TCMC,
								PORT:= TcMcGlobal.NCPORT_TCMC,
								IDXGRP:=TcMcGlobal.Axis.Parameter.IDXGRP+Axis.NcToPlc.AxisId,
								IDXOFFS:= TcMcGlobal.Axis.Parameter.IDXOFFS.VELOREFSEARCH,
								LEN:= SIZEOF(SearchVelocity),
								SRCADDR:= ADR(SearchVelocity),
								WRITE:= TRUE,
								TMOUT:= TcMcGlobal.tADSTimeOut);
		IF NOT fbAdsWriteParameter.Busy THEN
			IF fbAdsWriteParameter.Err	THEN
				Error := fbAdsWriteParameter.ERR;
				ErrorID := fbAdsWriteParameter.ERRID;
				iSubState := 0;
			ELSE
				IF Options.SyncDirection <> MC_Direction.MC_Undefined_Direction THEN
					iSubState := iSubState + 1;	(* Write homing sync direction *)
				ELSIF Options.SyncVelocity > 0.0 THEN
					iSubState := iSubState + 2;	(* Write homing sync velocity *)
				ELSIF Options.ReferenceMode <> E_EncoderReferenceMode.ENCODERREFERENCEMODE_DEFAULT THEN
					iSubState := iSubState + 3;	(* Write homing reference mode *)
				ELSE
					iSubState := 11; 	(* start homing (isubState = 11) *)
				END_IF
			END_IF
			fbAdsWriteParameter(WRITE:=FALSE);
		END_IF
	
	4: // Write homing sync direction
		SyncDirection := SEL(Options.SyncDirection = MC_Direction.MC_Positive_Direction, 1, 0);
		fbAdsWriteParameter(	NETID:= TcMcGlobal.NCNETID_TCMC,
								PORT:= TcMcGlobal.NCPORT_TCMC,
								IDXGRP:=TcMcGlobal.Axis.Parameter.IDXGRP+Axis.NcToPlc.AxisId,
								IDXOFFS:= TcMcGlobal.Axis.Parameter.IDXOFFS.ENCSYNCDIR,
								LEN:= SIZEOF(SyncDirection),
								SRCADDR:= ADR(SyncDirection),
								WRITE:= TRUE,
								TMOUT:= TcMcGlobal.tADSTimeOut);
		IF NOT fbAdsWriteParameter.Busy THEN
			IF fbAdsWriteParameter.Err	THEN
				Error := fbAdsWriteParameter.ERR;
				ErrorID := fbAdsWriteParameter.ERRID;
				iSubState := 0;
			ELSE
				IF Options.SyncVelocity > 0.0 THEN
					iSubState := iSubState + 1;	(* Write homing sync velocity *)
				ELSIF Options.ReferenceMode <> E_EncoderReferenceMode.ENCODERREFERENCEMODE_DEFAULT THEN
					iSubState := iSubState + 2;	(* Write homing reference mode *)
				ELSE
					iSubState := 11; 	(* start homing (isubState = 11) *)
				END_IF
			END_IF
			fbAdsWriteParameter(WRITE:=FALSE);
		END_IF
	
	5: // Write homing sync velocity
		SyncVelocity	:= Options.SyncVelocity;
		fbAdsWriteParameter(	NETID:= TcMcGlobal.NCNETID_TCMC,
								PORT:= TcMcGlobal.NCPORT_TCMC,
								IDXGRP:=TcMcGlobal.Axis.Parameter.IDXGRP+Axis.NcToPlc.AxisId,
								IDXOFFS:= TcMcGlobal.Axis.Parameter.IDXOFFS.VELOSYNCSEARCH,
								LEN:= SIZEOF(SyncVelocity),
								SRCADDR:= ADR(SyncVelocity),
								WRITE:= TRUE,
								TMOUT:= TcMcGlobal.tADSTimeOut);
		IF NOT fbAdsWriteParameter.Busy THEN
			IF fbAdsWriteParameter.Err	THEN
				Error := fbAdsWriteParameter.ERR;
				ErrorID := fbAdsWriteParameter.ERRID;
				iSubState := 0;
			ELSE
				IF Options.ReferenceMode <> E_EncoderReferenceMode.ENCODERREFERENCEMODE_DEFAULT THEN
					iSubState := iSubState + 1;	(* Write homing reference mode *)
				ELSE
					iSubState := 11; 	(* start homing (isubState = 11) *)
				END_IF
			END_IF
			fbAdsWriteParameter(WRITE:=FALSE);
		END_IF
	
	6: // Write homing reference mode
		ReferenceMode := Options.ReferenceMode;
		fbAdsWriteParameter(	NETID:= TcMcGlobal.NCNETID_TCMC,
								PORT:= TcMcGlobal.NCPORT_TCMC,
								IDXGRP:=TcMcGlobal.Axis.Parameter.IDXGRP+Axis.NcToPlc.AxisId,
								IDXOFFS:= TcMcGlobal.Axis.Parameter.IDXOFFS.ENCREFMODE,
								LEN:= SIZEOF(ReferenceMode),
								SRCADDR:= ADR(ReferenceMode),
								WRITE:= TRUE,
								TMOUT:= TcMcGlobal.tADSTimeOut);
		IF NOT fbAdsWriteParameter.Busy THEN
			IF fbAdsWriteParameter.Err	THEN
				Error := fbAdsWriteParameter.ERR;
				ErrorID := fbAdsWriteParameter.ERRID;
				iSubState := 0;
			ELSE
				iSubState := 11; 	(* start homing (isubState = 11) *)
			END_IF
			fbAdsWriteParameter(WRITE:=FALSE);
		END_IF
	
	11 :	(* start homing *)
		fbAdsWriteCmd(	NETID:= TcMcGlobal.NCNETID_TCMC,
						PORT:= TcMcGlobal.NCPORT_TCMC,
						IDXGRP:=TcMcGlobal.Axis.Functions.IDXGRP+Axis.NcToPlc.AxisId,
						IDXOFFS:= TcMcGlobal.Axis.Functions.IDXOFFS.CALIBR,
						LEN:= 0,
						SRCADDR:= 0,
						WRITE:= TRUE,
						TMOUT:= TcMcGlobal.tADSTimeOut);
		IF NOT fbAdsWriteCmd.Busy THEN
			IF fbAdsWriteCmd.ERR THEN
				Error := fbAdsWriteCmd.ERR;
				ErrorID := fbAdsWriteCmd.ERRID;
				iSubState := 0;
			ELSE
				fbTimeOut(IN:=TRUE, PT:=TcMcGlobal.tADSTimeOut);
				IF fbTimeOut.Q THEN
					(* calibration sequence did not start *)
					Error 	:= TRUE;
					ErrorID := MC_ERROR_CALIBRATION_ERROR; (* functional/calibration error *)
					iSubState := 0;
				END_IF;
				IF F_AxisIsCalibrating(StateDWord := Axis.NcToPlc.StateDWord) THEN
					(* calibration sequence started *)
					iState := STATE_RUNNING;
					iSubState := iSubState + 1; (* wait homing *)
				END_IF
			END_IF
		END_IF

	12 :	(* homing Busy *)
		(* wait for done in cyclic interface *)
		IF NOT F_AxisIsCalibrating(StateDWord := Axis.NcToPlc.StateDWord) THEN
			IF F_AxisIsCalibrated(StateDWord := Axis.NcToPlc.StateDWord) THEN
				Done 	:= TRUE;
			ELSE
				Error 	:= TRUE;
				ErrorID := MC_ERROR_CALIBRATION_ERROR; (* functional/calibration error *)
			END_IF;
			iSubState := 0;
		END_IF;
		IF F_AxisInErrorState(StateDWord := Axis.NcToPlc.StateDWord) THEN
			Done := FALSE;
			Error := TRUE;
			ErrorID := Axis.NcToPlc.ErrorCode; (* runtime errorcode *)
			iSubState := 0;
		END_IF;

	21 :	(* read homing position - 2009-04-17 KSt added *)
		fbAdsReadRefPos(	NETID:= TcMcGlobal.NCNETID_TCMC,
							PORT:= TcMcGlobal.NCPORT_TCMC,
							IDXGRP:=TcMcGlobal.Axis.Parameter.IDXGRP+Axis.NcToPlc.AxisId,
							IDXOFFS:= TcMcGlobal.Axis.Parameter.IDXOFFS.REF_POS,
							LEN:= SIZEOF(CalibrationValue),
							DESTADDR:= ADR(CalibrationValue),
							READ:= TRUE,
							TMOUT:= TcMcGlobal.tADSTimeOut);
		IF NOT fbAdsReadRefPos.Busy THEN
			IF fbAdsReadRefPos.Err	THEN
				Error := fbAdsReadRefPos.ERR;
				ErrorID := fbAdsReadRefPos.ERRID;
				iSubState := 0;
			ELSE
				fbSetPosition.Position := CalibrationValue;
				iSubState := iSubState + 1; (* set actual position *)
			END_IF
		END_IF

	22 :	(* Static Homing forcing position from user reference *)
		fbSetPosition.Options.ClearPositionLag:= Options.ClearPositionLag;	(* 2009-04-17 KSt - changed from TRUE to option flag*)
		fbSetPosition(
			Execute:= TRUE,
			(* Position:= Position, 2009-04-17 KSt - must be set before *)
			Mode:= FALSE,	(* absolute mode *)
			Axis:= Axis );
		IF fbSetPosition.Done THEN
			iSubState := 31;	(* set reference flag *)
		ELSIF NOT fbSetPosition.Busy THEN
			Error := TRUE;
			ErrorID := fbSetPosition.ErrorID;
			iSubState := 0;
		END_IF

	31 : 	(* Absolute homing - Set reference flag *)
		fbAdsWriteCmd(	NETID:= TcMcGlobal.NCNETID_TCMC,
						PORT:= AMSPORT_R0_NCSAF,
						IDXGRP:= TcMcGlobal.Axis.Functions.IDXGRP+Axis.NcToPlc.AxisId,
						IDXOFFS:= TcMcGlobal.Axis.Functions.IDXOFFS.SETCALFLAG,
						LEN:= SIZEOF(ReferenceFlagValue),
						SRCADDR:= ADR(ReferenceFlagValue),
						WRITE:= TRUE,
						TMOUT:= TcMcGlobal.tADSTimeOut );
		IF NOT fbAdsWriteCmd.Busy THEN
			Error := fbAdsWriteCmd.ERR;
			ErrorID := fbAdsWriteCmd.ERRID;
			Done := NOT Error;
			iSubState := 0;
		END_IF
		
	ELSE (* CASE : Unknown program state *)
		Error := TRUE;
		ErrorID := 16#FFFFFFFF;
		iSubState := 0;
END_CASE

ADSbusy := fbAdsWriteCmd.BUSY OR fbAdsWriteParameter.BUSY OR fbAdsReadRefPos.BUSY;

IF iSubState=0 THEN
	(* reset Busy immediately  when sequence ends *)
	IF Busy THEN
		LastExecutionResult.Done := Done;
		LastExecutionResult.CommandAborted := CommandAborted;
		LastExecutionResult.Error := Error;
		LastExecutionResult.ErrorID := ErrorID;
	END_IF
	Busy := FALSE;
ELSE
	(* copy calibration cam to interface *)
	Axis.PlcToNc.ControlDWord.5 := bCalibrationCam;
END_IF

Active := Busy;

END_FUNCTION_BLOCK

// POUs/Administrative/Axis Functions/MC_SetPosition
FUNCTION_BLOCK MC_SetPosition
(*
	This Function Block shifts the coordinate system of an axis by manipulating both 
	the set-point position as well as the actual position of an axis with the same value 
	without any movement caused. (Re-calibration with same following error).
	This can be used for instance for a reference situation. This Function Block can 
	also be used during motion without changing the commanded position, which is 
	now positioned in the shifted coordinate system.

	Note:
	Relative means that Position is added to the actual position value of the axis 
	at the time of execution. This results in a recalibration by a specified distance. 
	Absolute means that the actual position value of the axis is set to the value
	specified in the Position parameter.
*)
VAR_IN_OUT
	Axis				:	AXIS_REF; (*Reference to an axis*)
END_VAR
VAR_INPUT
	Execute				:	BOOL;	(* Start setting position in axis *)
	Position			:	LREAL;	(* Position unit [u] (Means Distance if Mode = RELATIVE) *)
	Mode (*Relative*)	: BOOL;		(* RELATIVE =True, ABSOLUTE = False (Default) *)
(* 	MC_ExecutionMode : ENUM *)		(* not available *)
	Options				:	ST_SetPositionOptions;	(* Beckhoff proprietary input *)
END_VAR
VAR_OUTPUT
	Done				:	BOOL;	(* Position has new value *)
	Busy				:	BOOL;	(* Shows that the Function Block is not finished *)
	Error				:	BOOL;	(* Signals that an error has occurred within the Function Block *)
{attribute 'displaymode':='hex'}
	ErrorID				:	UDINT;	(* Error identification *)
END_VAR
(*
	Note:
	RELATIVE means that Position is added to the actual position value of the axis 
	at the time of execution. This results in a recalibration by a specified distance. 
	ABSOLUTE means that the actual position value of the axis is set to the value 
	specified in the Position parameter.
	When changing the position on the fly, RELATIVE mode is supposed to be preferred
*)
VAR
	ADSbusy	: 	BOOL;
	stSetPos		:	_ST_TcNC_SetPosOnTheFly;
	iState		:	_E_TcMC_STATES := STATE_INITIALIZATION;
	fbAdsWrite	:	ADSWRITE;
END_VAR
VAR
{attribute 'conditionalshow'}
	fbOnTrigger	:	R_TRIG;
END_VAR


(*
	PlcOpen comment to MC_SetPosition
		The >Mode< input has later been renamed to >Relative<. Beckhoff cannot change the name for compatibility reasons.
		The input >MC_ExecutionMode<, defined by PlcOpen, is not implemented.
*)
IF NOT _F_TcMC_IsValidAxisRef(Axis) THEN // AXIS REFERENCE CHECK - 2020-09-17 KSt
	Error := TRUE;
	ErrorID := MC_ERROR_INVALIDREFERENCE;
	RETURN;
END_IF

fbOnTrigger(CLK:= Execute);

CASE iState OF
STATE_INITIALIZATION:
	Busy := FALSE;
	IF NOT Execute THEN
		Done := FALSE;
		Error := FALSE;			(* reset at falling edge of Execute *)
		ErrorID := 0;
	END_IF
	IF fbOnTrigger.Q THEN
		Busy := TRUE;
		(* initialize output values *)
		Done := FALSE;
		Error := FALSE;
		ErrorID := 0;
		fbAdsWrite(WRITE := FALSE);

		(* fill structure*)
		stSetPos.fNewActualPos := Position;
		stSetPos.nCtrlDWord.0 := SEL( Options.ClearPositionLag, FALSE, TRUE ); 		(* set bit 0 to clear the lag *)
		stSetPos.nCtrlDWord.1 := SEL( Options.SelectEncoderIndex, FALSE, TRUE ); 	(* set bit 1 to explicitly select an encoder / control loop - KSt 2009-04-09 *)
		stSetPos.nReserved[1]:=0;
		stSetPos.nReserved[2]:=0;

		IF Mode THEN
			(* relative mode *)
			stSetPos.nPosSetType := TCNC_POSSETTYPE_RELATIVE;
			stSetPos.fPreviousActualPos := 0;	(* value not used any longer since 2009-01-28 *)
		ELSE
			(* absolute mode *)
			stSetPos.nPosSetType := TCNC_POSSETTYPE_ABSOLUTE;
			stSetPos.fPreviousActualPos := Axis.NcToPlc.ActPos;	(* value not used any longer since 2009-01-28 *)
		END_IF

		IF Options.SelectEncoderIndex THEN (* KSt 2009-04-09 *)
			(* select the user defined encoder/control loop explicitly *)
			fbAdsWrite.IDXOFFS:= TcMcGlobal.Axis.Functions.IDXOFFS.SETPOSONTHEFLY + Options.EncoderIndex * 16#00100000;
		ELSE
			(* select the encoder / control loop that is defined by the AXIS_REF interface
				0  	=  select active encoder / control loop		- used when standard AXIS_REF interface is used
				1..n 	=  explicit encoder / control loop selection 	- used when dedicated encoder AXIS_REF interface is used 		*)
			fbAdsWrite.IDXOFFS:= TcMcGlobal.Axis.Functions.IDXOFFS.SETPOSONTHEFLY + Axis.NcToPlc.ControlLoopIndex * 16#00100000;
		END_IF

		fbAdsWrite(	NETID:= TcMcGlobal.NCNETID_TCMC,
					PORT:= AMSPORT_R0_NCSAF,
					IDXGRP:=TcMcGlobal.Axis.Functions.IDXGRP + Axis.NcToPlc.AxisId,
(*					IDXOFFS:= TcMcGlobal.Axis.Functions.IDXOFFS.SETPOSONTHEFLY + Options.EncoderIndex * 16#100000, *)(* add sub index - KSt 2008-10-22 *)
(*					IDXOFFS:= TcMcGlobal.Axis.Functions.IDXOFFS.SETPOSONTHEFLY, *)	(* see selection above - KSt 2009-04-09 *)
					LEN:= SIZEOF(stSetPos),
					SRCADDR:= ADR(stSetPos),
					WRITE:= TRUE,
					TMOUT:= TcMcGlobal.tADSTimeOut);
		iState := STATE_ORDER;
	END_IF;

STATE_ORDER:
	fbAdsWrite();
	IF NOT fbAdsWrite.Busy THEN
		IF fbAdsWrite.Err THEN
			ErrorID := fbAdsWrite.ErrId;
			Error := TRUE;
		ELSE
			Done := TRUE;
		END_IF;
		fbAdsWrite(WRITE := FALSE);
		iState := STATE_INITIALIZATION;
	END_IF;

ELSE  (* CASE : Unknown program state *)
	Error := TRUE;
	ErrorID := 16#FFFFFFFF;
	iState:= STATE_INITIALIZATION;
END_CASE

ADSbusy := fbAdsWrite.BUSY;

IF iState=STATE_INITIALIZATION THEN
	(* reset Busy immediately  when sequence ends *)
	Busy := FALSE;
END_IF

END_FUNCTION_BLOCK

// POUs/Motion/Superposition/MC_MoveSuperImposed
(*	MC_MovedSuperimposed	(extended version 2)

	This Function Block commands a controlled motion of a specified relative distance additional to an existing motion.
	The existing Motion is not interrupted, but is superimposed by the additional motion.

	- Version 2 adds multiple modes and feedback information to the 
	  standard MC_MoveSuperimposed block.
 	- The version 2 block is compatible to the MC_MovedSuperimposed block when Mode
	  SUPERPOSITIONMODE_VELOREDUCTION_ADDITIVEMOTION (integer value 1) is used.

	The values of Acceleration, Deceleration, and Jerk are additional values to the on-going motion, and not
	absolute ones. With this, the underlying FB always finishes its job in the same period of time regardless of
	whether a MC_MoveSuperimposed FB takes place concurrently.
 *)
FUNCTION_BLOCK MC_MoveSuperImposed
VAR_IN_OUT
	Axis				:	AXIS_REF; (*Reference to an axis*)
END_VAR
VAR_INPUT
	Execute			:	BOOL;	
	Mode 			:	E_SuperpositionMode;	
(*	ContinuousUpdate :	BOOL; *)		(* not available *)
	Distance			:	LREAL;		(* distance to catch up or fall back with the superposition process *)
	VelocityDiff		:	LREAL;		(* maximum velocity difference - will be added or subtrated to the process velocity *)
	Acceleration		:	LREAL;	
	Deceleration		:	LREAL;	
	Jerk				:	LREAL;		(* currently not used *)
	VelocityProcess	:	LREAL;		(* constant velocity of the axis without superposition *)
	Length			:	LREAL;		(* moved distance while the superposition takes place (name has been MaxDistance before) *)
	Options			:	ST_SuperpositionOptions;	
END_VAR
VAR_OUTPUT
	Done			:	BOOL;	
	Busy			:	BOOL;	
	Active			:	BOOL;	
	CommandAborted	:	BOOL;	
	Error			:	BOOL;	
{attribute 'displaymode':='hex'}
	ErrorID			:	UDINT;	
(*	CoveredDistance	:	LREAL;*)	(* not available *)
	Warning			: 	BOOL;	
	WarningId		: 	UDINT;	
	ActualVelocityDiff	: 	LREAL;		(* calculated maximum velocity boost during superposition <= VelocityDiff *)
	ActualDistance	: 	LREAL;		(* calculated superimposed distance <= Distance*)
	ActualLength		: 	LREAL;	(* calculated length of the superposition <= MaxDistance *)
	ActualAcceleration : 	LREAL;	(* calculated acceleration during superposition *)
	ActualDeceleration : 	LREAL;	(* calculated deceleration during superposition *)
END_VAR
VAR
	LastExecutionResult: 	_ST_FunctionBlockResults;
	ADSbusy		: 	BOOL;
	CompensationStarted: 	BOOL;
	AxisHasJobAtStartOfCompensation	: 	BOOL; 	(* HasJob flag when starting the compensation *)
	AxisIsMovingAtStartOfCompensation	:	BOOL; 	(* Moving flag when starting the compensation *)
	iState			: 	_E_TcMC_STATES := STATE_INITIALIZATION;
	fbAdsReadWrite	: 	ADSRDWRTEX;
	sNcCompensation	:	_ST_TcNC_Compensation2;
	// NCPORT_TCMC_SUPERPOSITION: UINT;		2021-10-19 KSt - constant removed (was here by mistake)
END_VAR
VAR
{attribute 'conditionalshow'}
	fbTrigger			:	R_TRIG;
{attribute 'conditionalshow'}
	fbTimeOut		: 	TON;
END_VAR

(* ====================================================================== *)
(* *)
(* ====================================================================== *)
fbTrigger(CLK:= Execute);

CASE iState OF
STATE_INITIALIZATION:	(* *)
	Busy := FALSE;
	Active := FALSE;

	IF NOT Execute THEN
		Done := FALSE;
		CommandAborted := FALSE;
		Error := FALSE;			(* reset at falling edge of Execute *)
		ErrorID := 0;
	END_IF;

    	IF fbTrigger.Q THEN
		(* initialize output values *)
		Done := FALSE;
		Busy := TRUE;
		CommandAborted := FALSE;
		Error := FALSE;
		ErrorID := 0;
		Warning := FALSE;
		WarningId := 0;
		LastExecutionResult.Done := FALSE;
		LastExecutionResult.CommandAborted := FALSE;
		LastExecutionResult.Error := FALSE;
		LastExecutionResult.ErrorID := 0;
		ActualVelocityDiff := 0;
		ActualDistance := 0;
		ActualLength := 0;
		CompensationStarted := FALSE;
		fbTimeOut(IN:= FALSE);
		fbAdsReadWrite(WRTRD:=FALSE);

		(* 2009-10-06 KSt - initial HasJob and InMotion state check *)
		AxisHasJobAtStartOfCompensation := F_AxisHasJob(Axis.NcToPlc.StateDWord);
		AxisIsMovingAtStartOfCompensation := F_AxisIsMoving(Axis.NcToPlc.StateDWord);
		(* error when ... *)
		(* 24.09.2009 HKP - Fehlerabfrage nur im Default-Fall mit  '(0) SUPERPOSITIONOPTION_ABORTATSTANDSTILL' sinnvoll *)
		(* IF  NOT F_AxisHasJob(Axis.NcToPlc.StateDWord) THEN  *) (* 12.6.2007 KSt - geändert von "NOT AxisIsMoving" nach "NOT AxisHasJob" *)
		IF  Options.AbortOption = SUPERPOSITIONOPTION_ABORTATSTANDSTILL AND NOT  F_AxisHasJob(Axis.NcToPlc.StateDWord) THEN
			ErrorID := MC_ERROR_AXIS_IS_NOT_MOVING;
			Error := TRUE;
		ELSE
			(* fill structure *)
			sNcCompensation.nCompType		:= Mode;
			sNcCompensation.fAccPlus		:= Acceleration;
			sNcCompensation.fAccMinus		:= Deceleration;
			sNcCompensation.fVeloDiff		:= VelocityDiff;
			sNcCompensation.fVeloProcess	:= VelocityProcess;
			sNcCompensation.fDistance		:= Distance;
			sNcCompensation.fLength		 	:= Length;
			(* WarningID holds optional parameters when sending the command to the NC *)
			sNcCompensation.nWarningId		:= Options.AbortOption; (* 2009-06-30 KSt *)

			(* fbAdsReadWrite.PORT := SEL(Axis.ADS.Port = 0, Axis.ADS.port, AMSPORT_R0_NCSAF);*)				(* KSt, 20140930 *) 
			fbAdsReadWrite.PORT := SEL(Axis.ADS.Port = 0, Axis.ADS.port, TcMcGlobal.NCPORT_TCMC_SUPERPOSITION);	(* KSt, 20140930 *)
			fbAdsReadWrite(NETID:= TcMcGlobal.NCNETID_TCMC,
							(* PORT:= TcMcGlobal.NCPORT_TCMC,*) 		(* KSt, 20090123 *)
							IDXGRP:= TcMcGlobal.Axis.Functions.IDXGRP+Axis.NcToPlc.AxisId,
							IDXOFFS:= TcMcGlobal.Axis.Functions.IDXOFFS.STARTSCOM,
							WRITELEN:= SIZEOF(sNcCompensation),
							READLEN:= SIZEOF(sNcCompensation),
							SRCADDR:= ADR(sNcCompensation),
							DESTADDR:= ADR(sNcCompensation),
							WRTRD:= TRUE,
							TMOUT:= TcMcGlobal.tADSTimeOut );

			iState := STATE_ORDER;
		END_IF;
	END_IF;

STATE_ORDER:  (* wait until command is accepted *)
	fbAdsReadWrite(WRTRD:= TRUE);
	IF NOT fbAdsReadWrite.Busy THEN
		IF fbAdsReadWrite.Err THEN
			Error := TRUE;
			ErrorID := fbAdsReadWrite.ErrId;
			iState := STATE_INITIALIZATION;
		ELSE
			IF fbAdsReadWrite.COUNT_R > 0 THEN
				ActualVelocityDiff := sNcCompensation.fVeloDiff;
				ActualDistance := sNcCompensation.fDistance;
				ActualLength := sNcCompensation.fLength;
				ActualAcceleration := sNcCompensation.fAccPlus;		(* 2010-02-25 KSt *)
				ActualDeceleration := sNcCompensation.fAccMinus;	(* 2010-02-25 KSt *)
				WarningId := sNcCompensation.nWarningId;	(* 2009-01-29 KSt *)
				Warning := WarningId <> 0;					(* 2009-01-29 KSt *)
			END_IF
			Active := TRUE;
			CompensationStarted := F_AxisIsCompensating(Axis.NcToPlc.StateDWord) ;
			iState := STATE_RUNNING;
		END_IF;
	END_IF;

STATE_RUNNING:  (* wait until axis stands still *)
	WarningId := sNcCompensation.nWarningId;
	Warning := WarningId <> 0;
(*	Busy := F_AxisIsCompensating(Axis.NcToPlc.StateDWord);
	IF Busy THEN	KSt, 29.4.2008 *)

	IF F_AxisIsCompensating(Axis.NcToPlc.StateDWord) THEN 	(* KSt, 29.4.2008 *)
		CompensationStarted := TRUE;
	ELSIF CompensationStarted  (* AND compensation finished now *) THEN
		IF AxisHasJobAtStartOfCompensation AND NOT F_AxisHasJob(Axis.NcToPlc.StateDWord) THEN (* 2009-10-06 KSt *)
			(* command aborted, move has been stopped before superposition finished because the HasJob flag turned off (KSt, 2009-08-13) *)
			CommandAborted := TRUE;
			iState := STATE_INITIALIZATION;
		ELSIF NOT AxisHasJobAtStartOfCompensation AND AxisIsMovingAtStartOfCompensation THEN (* 2009-10-06 KSt *)
			(* in case of axes coupled to actual position (encoder axes or disabled axes) *)
			IF NOT F_AxisIsMoving(Axis.NcToPlc.StateDWord) THEN (* 2009-10-06 KSt *)
				CommandAborted := TRUE;
				iState := STATE_INITIALIZATION;
			ELSE
				(* check moving state next cycle - delay is necessary since moving flag turnes off later than the compensation flag *)
				iState := STATE_WAITING;
			END_IF
		ELSE
			(* the initial HasJob or Moving state was the same as at end of compensation - assume that superposition completed *)
			Done := TRUE;
			iState := STATE_INITIALIZATION;
		END_IF
	ELSE (* compensation did not start so far *)
		(* check for superposition not beeing started (KSt, 12.01.2004) *)
		fbTimeOut(IN:= TRUE, PT:= T#50ms);
		IF fbTimeOut.Q THEN
			(*	when the ADS command comes back without any error but
				the compensation does not start anyway, we assume that  
				a very short compensation already has been executed. 
			*)
			Done := TRUE; (* after short timeout *)
			iState := STATE_INITIALIZATION;
		END_IF;
	END_IF

(* compensation not necessarily finished if axis stops (new modes available) - 2009-08-13 KSt *)
(*	IF NOT F_AxisHasJob(Axis.NcToPlc.StateDWord) THEN
		/* command aborted, move has been stopped before superposition finished (KSt, 12.01.2004) */
		CommandAborted := TRUE;
		iState := STATE_INITIALIZATION;
	END_IF
*)

STATE_WAITING : (* 2009-10-06 KSt  - state added for axes coupled to actual position (encoder axes or disabled axes) *)
	(* decide if superposition was completed or aborted in case of axes coupled to actual position (encoder axes or disabled axes) *)
	IF NOT F_AxisIsMoving(Axis.NcToPlc.StateDWord) THEN (* 2009-10-06 KSt *)
		(* command aborted, motion ended before superposition was finished because the axis is not moving any longer *)
		CommandAborted := TRUE;
	ELSE
		(* the initial HasJob or Moving state was the same as at end of compensation - assume that superposition completed *)
		Done := TRUE;
	END_IF
	CompensationStarted := FALSE;
	iState := STATE_INITIALIZATION;

ELSE  (* CASE : Unknown program state *)
	Error := TRUE;
	ErrorID := 16#FFFFFFFF;
	iState:= STATE_INITIALIZATION;
END_CASE

ADSbusy := fbAdsReadWrite.BUSY;
IF iState=STATE_INITIALIZATION THEN
	(* reset Busy immediately  when sequence ends *)
	IF Busy THEN
		LastExecutionResult.Done := Done;
		LastExecutionResult.CommandAborted := CommandAborted;
		LastExecutionResult.Error := Error;
		LastExecutionResult.ErrorID := ErrorID;
	END_IF
	Busy := FALSE;
	Active := FALSE;
END_IF

END_FUNCTION_BLOCK

// POUs/Administrative/Extensions/MC_SetOverride
FUNCTION_BLOCK MC_SetOverride
(*
	This Function Block sets the values of override for the whole axis, and all functions 
	that are working on that axis. The override parameters contribute as a factor to the 
	calculation of the commanded velocity, acceleration and jerk of the motion.
*)
VAR_IN_OUT
	Axis			:	AXIS_REF; (*Reference to an axis*)
END_VAR
VAR_INPUT
	Enable		:	BOOL;	
	VelFactor	:	LREAL		:= 1.0;	(* 1.0 = 100% *)
	AccFactor	:	LREAL		:= 1.0;	(* 1.0 = 100% *)	(* not supported *)
	JerkFactor	:	LREAL 		:= 1.0;	(* 1.0 = 100% *)	(* not supported *)
END_VAR
VAR_OUTPUT
	Enabled		:	BOOL;	
	Busy		:	BOOL;	
	Error		:	BOOL;	
{attribute 'displaymode':='hex'}
	ErrorID		:	UDINT;	
END_VAR
(*
	Notes:
	1. The Input AccFactor acts on positive and negative acceleration (deceleration).
	2. This Function Block sets the factor. The override factor is valid until a new override is set.
	3. The default values of the override factor are 1.0.
	4. The value of the overrides can be between 0.0 and 1.0. The behavior of values > 1.0 is 
	     vendor specific. Values< 0.0 are not allowed. The value 0.0 is not allowed for AccFactor 
	     and JerkFactor.
	5. The value 0.0 set to the VelFactor stops the axis without bringing it to the state Standstill.
	6. Override does not act on slave axes. (Axes in the state synchronized motion).
	7. The Function Block does not influence the state diagram of the axis.
	8. VelFactor can be changed at any time and acts directly on the ongoing motion.
	9. If in Discrete motion, reducing the AccFactor and/or JerkFactor can lead to a position 
	     overshoot  a possible cause of damage
	10. Activating this Function Block on an axis that is under control of MC_PositionProfile, 
	     MC_VelocityProfile, or MC_AccelerationProfile, is vendor specific.
*)
VAR
END_VAR


IF Enable THEN
	Busy := TRUE;
	IF VelFactor > 1 OR VelFactor < 0 THEN
		ErrorID := MC_ERROR_PARAMETER_NOT_CORRECT;
		Error := TRUE;
	ELSE
		Axis.PlcToNc.Override := LREAL_TO_UDINT(VelFactor*1000000);
		ErrorID := MC_ERROR_NO_ERROR;
		Error := FALSE;
		Enabled:=TRUE;
	END_IF;
ELSE
	Busy := FALSE;
	Enabled:=FALSE;
	Error := FALSE;			(* reset at falling edge of Execute *)
	ErrorID := 0;
END_IF;

END_FUNCTION_BLOCK

// POUs/Administrative/Axis Functions/MC_Reset
FUNCTION_BLOCK MC_Reset
(*
	This Function Block makes the transition from the state ErrorStop to StandStill
	or Disabled by resetting all internal axis-related errors. It does not affect the 
	output of the FB instances.
*)
VAR_IN_OUT
	Axis				:	AXIS_REF; (*Reference to an axis*)
END_VAR
VAR_INPUT
	Execute			:	BOOL;		(* B *)
END_VAR
VAR_OUTPUT
	Done			:	BOOL;		(* B *)
	Busy			:	BOOL;		(* E *)
	Error			:	BOOL;		(* B *)
{attribute 'displaymode':='hex'}
	ErrorID			:	UDINT;		(* B *)
END_VAR
VAR
	ADSbusy		: 	BOOL;
	iState			:	_E_TcMC_STATES := STATE_INITIALIZATION;
	LastExecutionResult: 	_ST_FunctionBlockResults;
END_VAR
VAR
{attribute 'hide'}
	fbAdsWrite		:	_TcMC_ADSWRITE;	(* 2010-05-31 KSt *)
(*	fbAdsWrite		:	ADSWRITE; *)		(* 2010-05-31 KSt *)
{attribute 'conditionalshow'}
	fbOnTrigger		:	R_TRIG;
END_VAR

IF NOT _F_TcMC_IsValidAxisRef(Axis) THEN // AXIS REFERENCE CHECK - 2020-09-17 KSt
	Error := TRUE;
	ErrorID := MC_ERROR_INVALIDREFERENCE;
	RETURN;
END_IF

fbOnTrigger(CLK:= Execute);

CASE iState OF
	STATE_INITIALIZATION: (* initial iState *)
		Busy := FALSE;
		IF NOT Execute THEN
			Done := FALSE;
			Error := FALSE;			(* reset at falling edge of Execute *)
			ErrorID := 0;
		END_IF
		IF fbOnTrigger.Q THEN
			Busy := TRUE;
			Done:= FALSE;
			Error := FALSE;
			ErrorID := 0;
(*			fbAdsWrite(WRITE:=FALSE);*)			(* 2010-05-31 KSt *)
			fbAdsWrite(WRITE:=FALSE, Axis:=Axis);	(* 2010-05-31 KSt *)

			fbAdsWrite(	NETID:= TcMcGlobal.NCNETID_TCMC,
						// PORT:= TcMcGlobal.NCPORT_TCMC,
						PORT:= TcMcGlobal.NCPORT_TCMC_RESET,	// 2021-10-19 KSt, changed to adjustable port number 
						IDXGRP:=TcMcGlobal.Axis.Functions.IDXGRP+Axis.NcToPlc.AxisId,
						IDXOFFS:= TcMcGlobal.Axis.Functions.IDXOFFS.RESET,
						LEN:= 0,
						SRCADDR:= 0 ,
						WRITE:=TRUE ,
						TMOUT:= TcMcGlobal.tADSTimeOut,
						Axis:=Axis		(* 2010-05-31 KSt *)
					);
			iState := STATE_ORDER;
		END_IF;

	STATE_ORDER:
(*		fbAdsWrite();*)			(* 2010-05-31 KSt *)
		fbAdsWrite( Axis:=Axis );	(* 2010-05-31 KSt *)
		 IF NOT fbAdsWrite.Busy THEN
			IF fbAdsWrite.Err THEN
				ErrorID := fbAdsWrite.ErrId;
				Error := TRUE;
			ELSE
				ErrorID := Axis.NcToPlc.ErrorCode;
				Error := ErrorID <> 0;
				Done := NOT Error;
			END_IF;
(*			fbAdsWrite(WRITE:=FALSE);*)			(* 2010-05-31 KSt *)
			fbAdsWrite(WRITE:=FALSE, Axis:=Axis );	(* 2010-05-31 KSt *)
			Axis.PlcToNc.PlcCycleControl.1 := 0; (* KSt - 2009-08 - reset exceeded flag for external set point generator *)
			iState := STATE_INITIALIZATION;
		END_IF

	ELSE  (* CASE : Unknown program state *)
		Error := TRUE;
		ErrorID := 16#FFFFFFFF;
		iState:= STATE_INITIALIZATION;
END_CASE;

ADSbusy := fbAdsWrite.BUSY;

IF iState=STATE_INITIALIZATION THEN
	(* reset Busy immediately  when sequence ends *)
	IF Busy THEN
		LastExecutionResult.Done := Done;
		LastExecutionResult.Error := Error;
		LastExecutionResult.ErrorID := ErrorID;
	END_IF
	Busy := FALSE;
END_IF

END_FUNCTION_BLOCK

// POUs/Administrative/External Set Point Generator/MC_ExtSetPointGenEnable
FUNCTION_BLOCK MC_ExtSetPointGenEnable
VAR_IN_OUT
	Axis	:	AXIS_REF; (*Reference to an axis*)
END_VAR
VAR_INPUT
	Execute : BOOL;
	Position : LREAL;
	PositionType : E_PositionType;
END_VAR
VAR_OUTPUT
	Done : BOOL;
	Busy: BOOL;
	Error: BOOL;
{attribute 'displaymode':='hex'}
	ErrorID: UDINT;
	Enabled: BOOL;
END_VAR
VAR
	LastExecutionResult	: 	_ST_FunctionBlockResults;
	iState				:	_E_TcMC_STATES := STATE_INITIALIZATION;
	ADSbusy			: 	BOOL;
	sExtSetPointGen 		: 	_ST_TcNC_SetPos;
	fbADSwrite			: 	ADSWRITE;
END_VAR
VAR
{attribute 'conditionalshow'}
	fbOnTrigger			: 	R_TRIG;
{attribute 'conditionalshow'}
	TimerStateFeedback	:	TON;
END_VAR

fbOnTrigger(CLK:= Execute);
Enabled := F_AxisHasExtSetPointGen(Axis.NcToPlc.StateDWord);

CASE iState OF
STATE_INITIALIZATION: (* initial iState *)
	Busy := FALSE;
	IF NOT Execute THEN
		Done := FALSE;
		Error := FALSE;
		ErrorID := 0;
	END_IF
	IF fbOnTrigger.Q THEN
		Busy := TRUE;
		(* initialization *)
		Done := FALSE;
		Error := FALSE;
		ErrorID := 0;
		LastExecutionResult.Done := FALSE;
		LastExecutionResult.CommandAborted := FALSE;
		LastExecutionResult.Error := FALSE;
		LastExecutionResult.ErrorID := 0;
		TimerStateFeedback(IN:=FALSE);
		fbADSwrite(WRITE:=FALSE);

		sExtSetPointGen.fNewPosIst:=Position;
		sExtSetPointGen.nPosIstType:=PositionType;
		fbADSwrite(	NETID:= TcMcGlobal.NCNETID_TCMC,
					PORT:=AMSPORT_R0_NCSAF,
					IDXGRP:= TcMcGlobal.Axis.Functions.IDXGRP + Axis.NcToPlc.AxisId,
					IDXOFFS:= TCMCGLOBAL.Axis.Functions.IDXOFFS.ENABLEEXTGEN,
					LEN:=SIZEOF(sExtSetPointGen),
					SRCADDR:=ADR(sExtSetPointGen),
					WRITE:=TRUE ,
					TMOUT:= TcMcGlobal.tADSTimeOut);
		iState := STATE_ORDER;
	END_IF

STATE_ORDER:  (* wait until command is accepted *)
	fbADSwrite(WRITE:= TRUE);
	IF NOT fbADSwrite.BUSY THEN
		Error := fbADSwrite.ERR;
		ErrorID := fbADSwrite.ERRID;
		IF NOT Error THEN
			IF F_AxisHasExtSetPointGen(Axis.NcToPlc.StateDWord) THEN
				Done := TRUE;
				Busy := FALSE;
				iState := STATE_INITIALIZATION;
			ELSE
				iState := STATE_RUNNING;
			END_IF
		ELSE
			Busy := FALSE;
			iState := STATE_INITIALIZATION;
		END_IF
		LastExecutionResult.Done := Done;
		LastExecutionResult.Error := Error;
		LastExecutionResult.ErrorID := ErrorID;
	END_IF

STATE_RUNNING: (* wait for feedback flag from StateDWord *)
	TimerStateFeedback(IN:=TRUE, PT:=t#50ms);
	IF F_AxisHasExtSetPointGen(Axis.NcToPlc.StateDWord) THEN
		Done := TRUE;
		Busy := FALSE;
		LastExecutionResult.Done := Done;
		LastExecutionResult.Error := Error;
		LastExecutionResult.ErrorID := ErrorID;
		iState := STATE_INITIALIZATION;
	ELSIF TimerStateFeedback.Q THEN
		(* the status flag 'external set point generator enabled' does not turn to TRUE *)
		Done := FALSE;
		Busy := FALSE;
		Error := TRUE;
		ErrorID := MC_ERROR_STATE_FEEDBACK_TIMEOUT;
		LastExecutionResult.Done := Done;
		LastExecutionResult.Error := Error;
		LastExecutionResult.ErrorID := ErrorID;
		iState := STATE_INITIALIZATION;
	END_IF
END_CASE

ADSbusy := fbAdsWrite.BUSY;

END_FUNCTION_BLOCK

// POUs/Administrative/External Set Point Generator/MC_ExtSetPointGenDisable
FUNCTION_BLOCK MC_ExtSetPointGenDisable
VAR_IN_OUT
	Axis	:	AXIS_REF; (*Reference to an axis*)
END_VAR
VAR_INPUT
	Execute : BOOL;
END_VAR
VAR_OUTPUT
	Done : BOOL;
	Busy: BOOL;
	Error: BOOL;
{attribute 'displaymode':='hex'}
	ErrorID: UDINT;
	Enabled: BOOL;
END_VAR
VAR
	LastExecutionResult	: 	_ST_FunctionBlockResults;
	iState				:	_E_TcMC_STATES := STATE_INITIALIZATION;
	ADSbusy			: 	BOOL;
	fbADSwrite			: 	ADSWRITE;
END_VAR
VAR
{attribute 'conditionalshow'}
	fbOnTrigger			: 	R_TRIG;
{attribute 'conditionalshow'}
	TimerStateFeedback	:	TON;
END_VAR

fbOnTrigger(CLK:= Execute);
Enabled := F_AxisHasExtSetPointGen(Axis.NcToPlc.StateDWord);

CASE iState OF
STATE_INITIALIZATION: (* initial iState *)
	Busy := FALSE;
	IF NOT Execute THEN
		Done := FALSE;
		Error := FALSE;
		ErrorID := 0;
	END_IF
	IF fbOnTrigger.Q THEN
		Busy := TRUE;
		(* initialization *)
		Done := FALSE;
		Error := FALSE;
		ErrorID := 0;
		LastExecutionResult.Done := FALSE;
		LastExecutionResult.CommandAborted := FALSE;
		LastExecutionResult.Error := FALSE;
		LastExecutionResult.ErrorID := 0;
		TimerStateFeedback(IN:=FALSE);
		fbADSwrite(WRITE:=FALSE);

		fbADSwrite(	NETID:= TcMcGlobal.NCNETID_TCMC,
					PORT:=AMSPORT_R0_NCSAF,
					IDXGRP:= TcMcGlobal.Axis.Functions.IDXGRP + Axis.NcToPlc.AxisId,
					IDXOFFS:= TCMCGLOBAL.Axis.Functions.IDXOFFS.DISABLEEXTGEN,
					LEN:=0,
					SRCADDR:=0,
					WRITE:=TRUE ,
					TMOUT:= TcMcGlobal.tADSTimeOut);
		iState := STATE_ORDER;
	END_IF

STATE_ORDER:  (* wait until command is accepted *)
	fbADSwrite(WRITE:= TRUE);
	IF NOT fbADSwrite.BUSY THEN
		Error := fbADSwrite.ERR;
		ErrorID := fbADSwrite.ERRID;
		IF NOT Error THEN
			IF NOT F_AxisHasExtSetPointGen(Axis.NcToPlc.StateDWord) THEN
				Done := TRUE;
				Busy := FALSE;
				iState := STATE_INITIALIZATION;
			ELSE
				iState := STATE_RUNNING;
			END_IF
		ELSE
			Busy := FALSE;
			iState := STATE_INITIALIZATION;
		END_IF
		Axis.PlcToNc.PlcCycleControl := 0; (* disable PLC cycle control *)
		LastExecutionResult.Done := Done;
		LastExecutionResult.Error := Error;
		LastExecutionResult.ErrorID := ErrorID;
	END_IF

STATE_RUNNING: (* wait for feedback flag from StateDWord *)
	TimerStateFeedback(IN:=TRUE, PT:=t#50ms);
	IF NOT F_AxisHasExtSetPointGen(Axis.NcToPlc.StateDWord) THEN
		Done := TRUE;
		Busy := FALSE;
		LastExecutionResult.Done := Done;
		LastExecutionResult.Error := Error;
		LastExecutionResult.ErrorID := ErrorID;
		iState := STATE_INITIALIZATION;
	ELSIF TimerStateFeedback.Q THEN
		(* the status flag 'external set point generator enabled' does not turn to TRUE *)
		Done := FALSE;
		Busy := FALSE;
		Error := TRUE;
		ErrorID := MC_ERROR_STATE_FEEDBACK_TIMEOUT;
		LastExecutionResult.Done := Done;
		LastExecutionResult.Error := Error;
		LastExecutionResult.ErrorID := ErrorID;
		iState := STATE_INITIALIZATION;
	END_IF
END_CASE

ADSbusy := fbAdsWrite.BUSY;

END_FUNCTION_BLOCK

// POUs/Administrative/Extensions/MC_OverrideFilter
FUNCTION_BLOCK MC_OverrideFilter
VAR_INPUT
	(* variables *)
	OverrideValueRaw		: DINT;
	(* parameter *)
	LowerOverrideThreshold	: DINT	:= 0;			(* 0...32767 digits *)
	UpperOverrideThreshold	: DINT	:= 32767;		(* 0...32767 digits *)
	OverrideSteps			: UDINT	:= 200;		(* 200 steps => 0.5 percent *)
	OverrideRecoveryTime	: TIME	:= T#150ms;	(* 150 ms *)
END_VAR
VAR_OUTPUT
	OverrideValueFiltered		: DWORD;			(* 0...1000000 counts *)
	OverridePercentFiltered	: LREAL;				(* 0...100 % *)
	Error					: BOOL;
{attribute 'displaymode':='hex'}
	ErrorID					: UDINT;
END_VAR
VAR
	bFirstCycle				: BOOL := TRUE;
	bThresholdActive			: BOOL := TRUE;
	InternalOverrideValueRaw	: DINT;
	LastOverrideValueRaw		: DINT := 16#FFFF;
	OverrideRange			: DINT;
END_VAR
VAR
{attribute 'conditionalshow'}
	fbTimer					: TON;
END_VAR

(* default value *)
Error	:= FALSE;
ErrorID	:= MC_ERROR_NO_ERROR;

(* check parameter / error handling:   'UpperOverrideThreshold > LowerOverrideThreshold'  AND  'OverrideSteps > 1'  *)
IF( (LowerOverrideThreshold >= UpperOverrideThreshold) OR (OverrideSteps <= 1) )THEN
	OverrideValueFiltered		:= 0;
	OverridePercentFiltered	:= 0.0;
	Error	:= TRUE;
	ErrorID	:= MC_ERROR_PARAMETER_NOT_CORRECT;
	RETURN;
END_IF;

(* first cycle: timer must be elapsed *)
IF ( bFirstCycle ) THEN
	fbTimer( IN:=TRUE, PT:= T#0s );
	bFirstCycle := FALSE;
END_IF;

IF ( OverrideValueRaw >= UpperOverrideThreshold ) THEN
	InternalOverrideValueRaw := UpperOverrideThreshold;
	bThresholdActive := TRUE;
ELSIF ( OverrideValueRaw <= LowerOverrideThreshold ) THEN
	InternalOverrideValueRaw := LowerOverrideThreshold;
	bThresholdActive := TRUE;
ELSE
	InternalOverrideValueRaw := OverrideValueRaw;
	bThresholdActive := FALSE;
END_IF;

fbTimer( IN:=TRUE, PT:= OverrideRecoveryTime );
IF( fbTimer.Q = TRUE OR bThresholdActive )THEN
	OverrideRange := UpperOverrideThreshold - LowerOverrideThreshold;
(*	IF (  bThresholdActive OR ABS( InternalRawOverrideValue - LastRawOverrideValue ) >= (0.5 * OverrideRange / OverrideSteps)  ) THEN *)
(*	IF (  bThresholdActive OR ABS( InternalOverrideValueRaw - LastOverrideValueRaw ) >= ( OverrideRange / OverrideSteps)  ) THEN*)
	IF (  bThresholdActive OR ABS( InternalOverrideValueRaw - LastOverrideValueRaw ) >= ( OverrideRange / UDINT_TO_DINT(OverrideSteps))  ) THEN (* 20110511 KSt type conversion for TC3 *)
		OverrideValueFiltered := DINT_TO_DWORD(((InternalOverrideValueRaw - LowerOverrideThreshold) * 1000 / OverrideRange) * 1000);
		OverridePercentFiltered := DWORD_TO_LREAL( OverrideValueFiltered ) * LREAL#0.0001;
		LastOverrideValueRaw := InternalOverrideValueRaw;
		fbTimer( IN:=FALSE, PT:= OverrideRecoveryTime );
	END_IF;
END_IF;

END_FUNCTION_BLOCK

// POUs/Administrative/Status and Parameter/MC_ReadStatus
FUNCTION_BLOCK MC_ReadStatus
(*	This Function Block returns in detail the status of the axis with respect to the motion currently in progress *)
VAR_IN_OUT
	Axis				:	AXIS_REF; (*Reference to an axis*)
END_VAR
VAR_INPUT
	Enable			:	BOOL;	
END_VAR
VAR_OUTPUT
	Valid			:	BOOL;	
	Busy			: 	BOOL;	
	Error			:	BOOL;	
{attribute 'displaymode':='hex'}
	ErrorID			:	UDINT;	
	(* motion control statemachine states: *)
	ErrorStop		:	BOOL;	
	Disabled			:	BOOL;	
	Stopping			:	BOOL;	
	StandStill		:	BOOL;	
	DiscreteMotion	:	BOOL;	
	ContinuousMotion	:	BOOL;	
	SynchronizedMotion:	BOOL;	
	Homing			:	BOOL;
	(* additional status *)
	ConstantVelocity	:	BOOL;	
	Accelerating		:	BOOL;	
	Decelerating		:	BOOL;	
	(* status data structure *)
	Status			: 	ST_AxisStatus;	
END_VAR
VAR
END_VAR

IF NOT _F_TcMC_IsValidAxisRef(Axis) THEN // AXIS REFERENCE CHECK - 2020-09-17 KSt
	Error := TRUE;
	ErrorID := MC_ERROR_INVALIDREFERENCE;
	RETURN;
END_IF

IF Enable THEN
	Busy := TRUE;

		Axis.ReadStatus();
	Status := Axis.Status;

	Error			:= 	Status.Error;
	ErrorID			:= 	Status.ErrorID;

	(* motion control statemachine states: *)
	ErrorStop		:= 	Status.ErrorStop;
	Disabled			:= 	Status.Disabled;
	Stopping			:= 	Status.Stopping;
	StandStill		:= 	Status.StandStill;
	DiscreteMotion	:= 	Status.DiscreteMotion;
	ContinuousMotion	:= 	Status.ContinuousMotion;
	SynchronizedMotion:= 	Status.SynchronizedMotion;
	Homing			:= 	Status.Homing;

	(* additional status *)
	ConstantVelocity	:= 	Status.ConstantVelocity;
	Accelerating		:= 	Status.Accelerating;
	Decelerating		:= 	Status.Decelerating;

	Valid := TRUE;
ELSE
	Busy := FALSE;
	Valid := FALSE;
	Error := FALSE;	(* reset at falling edge of Execute *)
	ErrorID := 0;
END_IF

END_FUNCTION_BLOCK

// POUs/Administrative/External Set Point Generator/MC_ExtSetPointGenFeed
FUNCTION MC_ExtSetPointGenFeed : BOOL

VAR_INPUT
	Position		: LREAL;
	Velocity		: LREAL;
	Acceleration	: LREAL;
	Direction 	: DINT;
END_VAR
VAR
	GetTaskIndex : GETCURTASKINDEX;
END_VAR

(*All VAR_IN_OUT variables have been moved to the end of the declaration due to compatibility reasons*)
VAR_IN_OUT
	Axis	:	AXIS_REF; (*Reference to an axis*)
END_VAR

Axis.PlcToNc.ExtSetPos := Position;
Axis.PlcToNc.ExtSetVelo := Velocity;
Axis.PlcToNc.ExtSetAcc := Acceleration;
Axis.PlcToNc.ExtSetDirection := Direction;	(* 24-05-2012 KST - type cast DINT_TO_UDINT entfernt *) 

GetTaskIndex();
Axis.PlcToNc.PlcCycleControl.0 := 1; (* activate PLC cycle information to NC *)
Axis.PlcToNc.PlcCycleControl.1 := TwinCAT_SystemInfoVarList._TaskInfo[ GetTaskIndex.index ].cycleTimeExceeded;
Axis.PlcToNc.PlcCycleCount := Axis.PlcToNc.PlcCycleCount + 1;

END_FUNCTION

// POUs/Administrative/Status and Parameter/MC_ReadBoolParameter
FUNCTION_BLOCK MC_ReadBoolParameter
(*	This Function Block returns the value of a vendor specific boolean parameter.*)
VAR_IN_OUT
	Axis				:	AXIS_REF; (*Reference to an axis*)
END_VAR
VAR_INPUT
	Enable				:	BOOL;		
	ParameterNumber		:	MC_AxisParameter; // 2023-03 KSt changed from INT to MC_AxisParameter		
	ReadMode			:	E_ReadMode	:= ReadMode_Once;	 (* Beckhoff proprietary input *)
END_VAR
VAR_OUTPUT
	Valid				:	BOOL;	
	Busy				: 	BOOL;	
	Error				:	BOOL;	
{attribute 'displaymode':='hex'}
	ErrorID				:	UDINT;
	Value				:	BOOL;	
END_VAR
VAR
	ADSbusy: BOOL;
	fbReadWriteParameter: 	_FB_ReadWriteParameter;
END_VAR
VAR
//{attribute 'conditionalshow'}
//	nParatype 			: 	_E_ParameterType;	(* removed 2021-04-12 KSt - not required *)
{attribute 'conditionalshow'}
	dwValue 			: 	DWORD;
{attribute 'conditionalshow'}
	lrValue				: 	LREAL;
{attribute 'conditionalshow'}
	bStarted			:	BOOL;
{attribute 'conditionalshow'}
	fbTrigger 			: 	R_TRIG;
END_VAR

IF NOT Enable THEN
	Valid := FALSE;
	Error := FALSE;			(* reset at falling edge of Execute *)
	ErrorID := 0;
END_IF
IF ReadMode = ReadMode_Once THEN
	fbTrigger(CLK:= Enable);
	IF fbTrigger.Q AND NOT bStarted THEN
		bStarted := TRUE;
		Valid := FALSE;
		Error := FALSE;
		ErrorID := MC_ERROR_NO_ERROR;
	END_IF;
ELSE
	IF Enable AND NOT bStarted THEN
		bStarted := TRUE;
		Valid := FALSE;
		Error := FALSE;
		ErrorID := MC_ERROR_NO_ERROR;
	END_IF;
END_IF;
(* *)
IF bStarted THEN
//	nParatype := PARAMETERTYPE_BOOL;
	fbReadWriteParameter.ParameterPointer := 0;
	fbReadWriteParameter.ParameterSize := 0;
	fbReadWriteParameter(Enable:= TRUE, ParameterNumber:= ParameterNumber, Mode:= READWRITEPARAMETERMODE_READ,
						(*ParameterType:=nParatype,*) Axis:= Axis, ValueLreal:= lrValue, ValueDword := dwValue, ValueBool := Value);
	IF fbReadWriteParameter.Done THEN
		bStarted := FALSE;
		Valid := TRUE;
		fbReadWriteParameter(Enable:= FALSE, ParameterNumber:= ParameterNumber, Mode:= READWRITEPARAMETERMODE_READ,
						(*ParameterType:= nParatype,*) Axis:= Axis, ValueLreal:= lrValue, ValueDword := dwValue, ValueBool := Value);
	END_IF;
	IF fbReadWriteParameter.Error THEN
		bStarted := FALSE;
		Valid := FALSE;
		Error := TRUE;
		ErrorID := fbReadWriteParameter.ErrorID;
		fbReadWriteParameter(Enable:= FALSE, ParameterNumber:= ParameterNumber, Mode:= READWRITEPARAMETERMODE_READ,
						(*ParameterType:= nParatype,*) Axis:= Axis, ValueLreal:= lrValue, ValueDword := dwValue, ValueBool := Value);
	END_IF;
END_IF;

ADSbusy := fbReadWriteParameter.ADSbusy;
Busy := (Enable AND ReadMode<>ReadMode_Once) OR bStarted;

END_FUNCTION_BLOCK

// POUs/Motion/Point To Point Motion/MC_MoveModulo
FUNCTION_BLOCK MC_MoveModulo
(* This Function Block commands a controlled motion to a specified absolute modulo position. *)
VAR_IN_OUT
	Axis				:	AXIS_REF; (*Reference to an axis*)
END_VAR
VAR_INPUT
	Execute			:	BOOL;
	Position			:	LREAL;
	Velocity			:	LREAL;
	Acceleration		:	LREAL;
	Deceleration		:	LREAL;
	Jerk				:	LREAL;
	Direction			:	MC_Direction;	(* E *)	(* modulo shortest way, modulo positive, modulo negative *)
	BufferMode		:	MC_BufferMode;(* E *)
	Options			: 	ST_MoveOptions;
END_VAR
VAR_OUTPUT
	Done				:	BOOL;	
	Busy				: 	BOOL;	
	Active				: 	BOOL;	
	CommandAborted		:	BOOL;	
	Error				:	BOOL;	
{attribute 'displaymode':='hex'}
	ErrorID				:	UDINT;	
END_VAR
VAR
	LastExecutionResult: _ST_FunctionBlockResults;
	ADSbusy: BOOL;
	MoveGeneric: _FB_MoveUniversalGeneric;
(*	StartType: UDINT;*)
	StartType: _E_TcNC_StartPosType;	(* 20110511 KSt type changed for TC3 *)
	CmdNo: UINT;
	TriggerExecute: R_TRIG;
END_VAR


(*  new move modulo code - KST 2012-03-23 *)
TriggerExecute(CLK:=Execute);
IF NOT Execute THEN // Reset Error when called with Execute = FALSE FAP 2022-02-28
	Error := FALSE;
	ErrorID := 0;
	Done := FALSE;
	Busy := FALSE;
	Active := FALSE;
	CommandAborted := FALSE;
ELSIF TriggerExecute.Q AND NOT MoveGeneric.Busy THEN
// IF TriggerExecute.Q AND NOT MoveGeneric.Busy THEN	
	(* initialize the start type when block is triggered *)
	CASE Direction OF
		MC_Positive_Direction:
			StartType := TCNC_START_MODULO_PLUS;
		MC_Shortest_Way:
			StartType := TCNC_START_MODULO_SHORT;
		MC_Negative_Direction:
			StartType := TCNC_START_MODULO_MINUS;
		MC_Current_Direction:
			StartType := TCNC_START_MODULO_CURRENT;
		ELSE
			StartType := 0; (* set to undefined *)
			Error := TRUE;
			ErrorID := MC_ERROR_WRONG_MODE;
			Done := FALSE;
			Busy := FALSE;
			Active := FALSE;
			CommandAborted := FALSE;
			(* generic move block will not be called *)
	END_CASE
END_IF

IF StartType<>0 THEN
	(* just call the generic move block *)
	MC_MoveModuloCall();
END_IF


(* old code before 2012-03-23 - KST *)
(*
CASE Direction OF
	MC_Positive_Direction:
		StartType := TCNC_START_MODULO_PLUS;
		MC_MoveModuloCall();

	MC_Shortest_Way:
		StartType := TCNC_START_MODULO_SHORT;
		MC_MoveModuloCall();

	MC_Negative_Direction:
		StartType := TCNC_START_MODULO_MINUS;
		MC_MoveModuloCall();

	MC_Current_Direction:
		StartType := TCNC_START_MODULO_CURRENT;
		MC_MoveModuloCall();
	ELSE
		IF Execute THEN
			Error := TRUE;
			ErrorID := MC_ERROR_WRONG_MODE;
		ELSE
			Error := FALSE;
			ErrorID := 0;
		END_IF
		Execute := FALSE;
		MC_MoveModuloCall();
		Done := FALSE;
		Busy := FALSE;
		Active := FALSE;
		CommandAborted := FALSE;
END_CASE
*)

ACTION MC_MoveModuloCall:
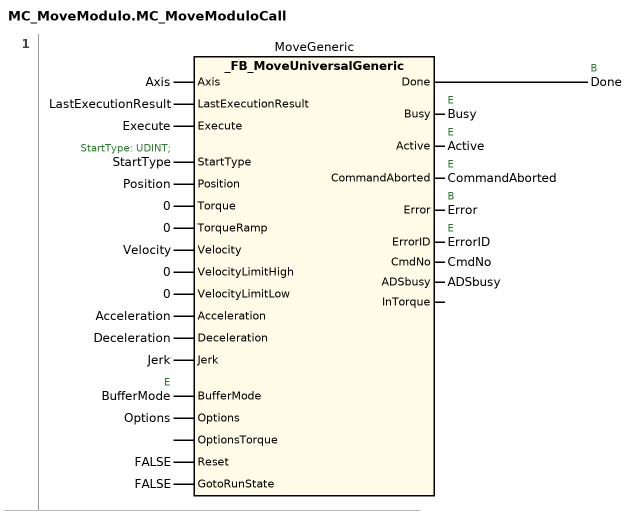
// NETWORK 1
//   StartType: StartType: UDINT;
//   BufferMode: E
//   Busy: E
//   Active: E
//   CommandAborted: E
//   Error: B
//   ErrorID: E
//   Done: B
MoveGeneric(
    Axis := Axis,
    LastExecutionResult := LastExecutionResult,
    Execute := Execute,
    StartType := StartType,
    Position := Position,
    Torque := 0,
    TorqueRamp := 0,
    Velocity := Velocity,
    VelocityLimitHigh := 0,
    VelocityLimitLow := 0,
    Acceleration := Acceleration,
    Deceleration := Deceleration,
    Jerk := Jerk,
    BufferMode := BufferMode,
    Options := Options,
    Reset := FALSE,
    GotoRunState := FALSE,
    Busy => Busy,
    Active => Active,
    CommandAborted => CommandAborted,
    Error => Error,
    ErrorID => ErrorID,
    CmdNo => CmdNo,
    ADSbusy => ADSbusy); // _FB_MoveUniversalGeneric
Done := MoveGeneric.Done;
END_ACTION

END_FUNCTION_BLOCK

// POUs/Motion/Point To Point Motion/MC_MoveVelocity
FUNCTION_BLOCK MC_MoveVelocity
(*	This Function Block commands a never ending controlled motion at a specified velocity. *)
VAR_IN_OUT
	Axis				:	AXIS_REF; (*Reference to an axis*)
END_VAR
VAR_INPUT
	Execute			:	BOOL;	
(*	ContinuousUpdate :	BOOL; *)	(* not available *)
	Velocity			:	LREAL;	
	Acceleration		:	LREAL;	
	Deceleration		:	LREAL;	
	Jerk				:	LREAL;	
	Direction			:	MC_Direction := MC_Positive_Direction;
	BufferMode		:	MC_BufferMode;	
	Options			: 	ST_MoveOptions; 
END_VAR
VAR_OUTPUT
	InVelocity		:	BOOL;		(* Commanded velocity reached *)
	Busy			: 	BOOL;	
	Active			: 	BOOL;	
	CommandAborted	:	BOOL;	
	Error			:	BOOL;	
{attribute 'displaymode':='hex'}
	ErrorID			:	UDINT;	
END_VAR
VAR
	LastExecutionResult: 	_ST_FunctionBlockResults;
	ADSbusy		: 	BOOL;
	MoveGeneric		: 	_FB_MoveUniversalGeneric;
	CmdNo: UINT;
END_VAR

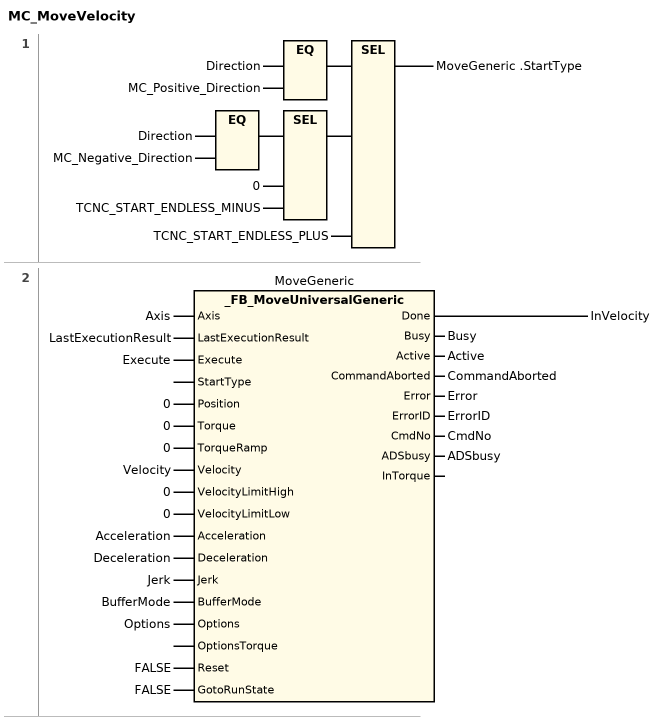
// NETWORK 1
MoveGeneric .StartType := SEL(Direction = MC_Positive_Direction, SEL(Direction = MC_Negative_Direction, 0, TCNC_START_ENDLESS_MINUS), TCNC_START_ENDLESS_PLUS);

// NETWORK 2
MoveGeneric(
    Axis := Axis,
    LastExecutionResult := LastExecutionResult,
    Execute := Execute,
    Position := 0,
    Torque := 0,
    TorqueRamp := 0,
    Velocity := Velocity,
    VelocityLimitHigh := 0,
    VelocityLimitLow := 0,
    Acceleration := Acceleration,
    Deceleration := Deceleration,
    Jerk := Jerk,
    BufferMode := BufferMode,
    Options := Options,
    Reset := FALSE,
    GotoRunState := FALSE,
    Busy => Busy,
    Active => Active,
    CommandAborted => CommandAborted,
    Error => Error,
    ErrorID => ErrorID,
    CmdNo => CmdNo,
    ADSbusy => ADSbusy); // _FB_MoveUniversalGeneric
InVelocity := MoveGeneric.Done;

END_FUNCTION_BLOCK

// POUs/Administrative/Status and Parameter/MC_ReadParameter
FUNCTION_BLOCK MC_ReadParameter
(*	This Function Block returns the value of a vendor specific parameter *)
VAR_IN_OUT
	Axis				:	AXIS_REF; (*Reference to an axis*)
END_VAR
VAR_INPUT
	Enable			:	BOOL;		
	ParameterNumber	:	MC_AxisParameter; // 2023-03 KSt changed from INT to MC_AxisParameter		
	ReadMode		:	E_ReadMode := ReadMode_Once;	 (* Beckhoff proprietary input *)
END_VAR
VAR_OUTPUT
	Valid			:	BOOL;		
	Busy			: 	BOOL;		
	Error			:	BOOL;		
{attribute 'displaymode':='hex'}
	ErrorID			:	UDINT;		
	Value			:	LREAL;		
END_VAR
VAR
	ADSbusy		: 	BOOL;
	fbReadWriteParameter: 	_FB_ReadWriteParameter;
END_VAR
VAR
//{attribute 'conditionalshow'}
//	nParatype 		: 	_E_ParameterType;	(* removed 2021-04-12 KSt - not required *)
{attribute 'conditionalshow'}
	dwValue 			: 	DWORD;
{attribute 'conditionalshow'}
	bValue 			: 	BOOL;
{attribute 'conditionalshow'}
	bStarted			:	BOOL;
{attribute 'conditionalshow'}
	fbTrigger		 	: 	R_TRIG;
END_VAR

(* ====================================================================== *)
(* *)
(* ====================================================================== *)
IF NOT Enable THEN
	Valid := FALSE;
	Error := FALSE;			(* reset at falling edge of Execute - just ErrorID will be kept til next rising edge *)
	ErrorID := 0;
END_IF
IF ReadMode = ReadMode_Once THEN
	fbTrigger(CLK:= Enable);
	IF fbTrigger.Q AND NOT bStarted THEN
		Value := 0;
		bStarted := TRUE;
		Valid := FALSE;
		Error := FALSE;
		ErrorID := MC_ERROR_NO_ERROR;
	END_IF;
ELSE
	IF Enable AND NOT bStarted THEN
		bStarted := TRUE;
		Valid := FALSE;
		Error := FALSE;
		ErrorID := MC_ERROR_NO_ERROR;
	END_IF;
	IF NOT Enable AND NOT bStarted THEN
		Valid := FALSE;
		Error := FALSE;
		ErrorID := MC_ERROR_NO_ERROR;
	END_IF;
END_IF;

IF bStarted THEN
//	nParatype := PARAMETERTYPE_LREAL;
	fbReadWriteParameter.ParameterPointer := 0;
	fbReadWriteParameter.ParameterSize := 0;
	fbReadWriteParameter(Enable:= TRUE, ParameterNumber:= ParameterNumber, Mode:= READWRITEPARAMETERMODE_READ,
						(*ParameterType:=nParatype,*) Axis:= Axis, ValueLreal:= Value, ValueDword := dwValue, ValueBool := bValue);
	IF fbReadWriteParameter.Done THEN
		bStarted := FALSE;
		Valid := TRUE;
		fbReadWriteParameter(Enable:= FALSE, ParameterNumber:= ParameterNumber, Mode:= READWRITEPARAMETERMODE_READ,
						(*ParameterType:= nParatype,*) Axis:= Axis, ValueLreal:= Value, ValueDword := dwValue, ValueBool := bValue);
	END_IF;
	IF fbReadWriteParameter.Error THEN
		Value := 0;
		bStarted := FALSE;
		Valid := FALSE;
		Error := TRUE;
		ErrorID := fbReadWriteParameter.ErrorID;
		fbReadWriteParameter(Enable:= FALSE, ParameterNumber:= ParameterNumber, Mode:= READWRITEPARAMETERMODE_READ,
						(*ParameterType:= nParatype,*) Axis:= Axis, ValueLreal:= Value, ValueDword := dwValue, ValueBool := bValue);
	END_IF;
END_IF;

ADSbusy := fbReadWriteParameter.ADSbusy;
Busy := (Enable AND ReadMode<>ReadMode_Once) OR bStarted;

END_FUNCTION_BLOCK

// POUs/Administrative/Touch Probe/MC_TouchProbe
FUNCTION_BLOCK MC_TouchProbe
(*	The function block is used to record an axis position at a trigger event *)
VAR_IN_OUT
	Axis				:	AXIS_REF; (*Reference to an axis*)
	TriggerInput		: 	TRIGGER_REF; 	(* Reference to the trigger signal source. *)
END_VAR
VAR_INPUT
	Execute			:	BOOL;		(* Starts touch probe recording *)
	WindowOnly		: 	BOOL;		(* Enables the monitoring window *)
	FirstPosition		: 	LREAL;	(* Beginning of the monitoring window *)
	LastPosition		: 	LREAL;	(* Ending of the monitoring window *)
END_VAR
VAR_OUTPUT
	Done			:	BOOL;		(* move completed *)
	Busy			: 	BOOL;		(* function block is currently Busy *)
	CommandAborted	: 	BOOL;	
	Error			:	BOOL;		(* Signals that error has occurred within Function Block *)
{attribute 'displaymode':='hex'}
	ErrorID			:	UDINT;		(* Error identification *)
	RecordedPosition	:	LREAL;	(* Position where trigger event occurred *)
	RecordedData	:	MC_TouchProbeRecordedData;	(* data additional to RecordedPosition *)
END_VAR
VAR
	ADSbusy: BOOL;
	iState			: 	_E_TcMC_STATES := STATE_INITIALIZATION;
	ExternalLatchValid: BOOL;
	TouchProbeValid	: 		ARRAY[1..4] OF UDINT;	(* valid state of probes 1..4 *)
	TouchProbeActive: 		ARRAY[1..4] OF UDINT;	(* activation state of probes 1..4 *)
	TouchProbeValue : 		ARRAY[1..4] OF LREAL;	(* last recorded value of probes 1..4 *)
	TouchProbeModuloValue : 	ARRAY[1..4] OF LREAL;	(* last recorded modulo value of probes 1..4 *)
	TouchProbeCounter : 		ARRAY[1..4] OF UDINT;	(* last recorded value counter of probes 1..4 *)
	TouchProbeInactiveCounter: 	ARRAY[1..4] OF INT;	(* number of cycles where the probes 1..4 where inactive (activation monitoring) *)
	stTouchProbeActivation : _ST_TcNc_TouchProbeActivation;
	stTouchProbeStatusRequest : _ST_TcNc_TouchProbeStatusRequest;
	stTouchProbeStatusResponse : _ST_TcNc_TouchProbeStatusResponse;
	stTouchProbeDeactivation : _ST_TcNc_TouchProbeDeactivation;
END_VAR
VAR
{attribute 'conditionalshow'}
	LastTouchProbeValue : 	ARRAY[1..4] OF LREAL;	(* last recorded value of probes 1..4 *)
{attribute 'conditionalshow'}
	LastTouchProbeCounter : 	ARRAY[1..4] OF UDINT;	(* last recorded value counter of probes 1..4 *)
{attribute 'conditionalshow'}
	fbADSwrite		: 	ADSWRITE;
{attribute 'conditionalshow'}
	fbAdsReadValid	: 	ADSREAD;
{attribute 'conditionalshow'}
	fbAdsReadValue	: 	ADSREAD;
{attribute 'conditionalshow'}
	fbAdsReadState	: 	ADSREAD;
{attribute 'conditionalshow'}
	fbAdsReadModulo: 	ADSREAD;
{attribute 'conditionalshow'}
	fbAdsReadLatchStatus: ADSRDWRTEX;
{attribute 'conditionalshow'}
	TimerAdsReadState: 	TON;
{attribute 'conditionalshow'}
	RtrigPlcEvent		: 	R_TRIG;
{attribute 'conditionalshow'}
	FtrigPlcEvent		: 	F_TRIG;
{attribute 'conditionalshow'}
	fbOnTrigger		: 	R_TRIG;
{attribute 'conditionalshow'}
	Restart			: 	BOOL;	(* restart probe sequence when the trigger was outside the defined window *)
{attribute 'conditionalshow'}
	InWindow		: 	BOOL;	(* probe value is inside the defined window *)
{attribute 'conditionalshow'}
	ModuloFactor		: 	LREAL;	(* axis' modulo factor read from the NC *)
{attribute 'conditionalshow'}
	tempModuloFactor	: 	LREAL;	(* axis' modulo factor read from the NC - used in ADS call *)
{attribute 'conditionalshow'}
	InitDone			: 	BOOL;	(* initialization on start-up finished *)
{attribute 'conditionalshow'}
	IndexOffset		: 	WORD;
{attribute 'conditionalshow'}
	iTriggerInput		: 	TRIGGER_REF; 	(* B *)	(* Reference to the trigger signal source. *)
{attribute 'conditionalshow'}
	i: INT;
END_VAR


(* 	MC_TouchProbe main sequence *)

fbOnTrigger(CLK:= Execute);
ExternalLatchValid := F_AxisExternalLatchValid(Axis.NcToPlc.StateDWord);

CASE iState OF
	STATE_INITIALIZATION :
		Busy := FALSE;
		IF NOT Execute THEN
			Done := FALSE;
			Error := FALSE;			(* reset at falling edge of Execute *)
			ErrorID := 0;
		END_IF

		ActTouchProbeStartupInit();	(* will return InitDone *)

		(* read version of NC *)
		IF TcMcGlobal.NcDeviceInfoNcVersion=0 THEN
			TcMcGlobal.ReadDeviceInfo();
		END_IF
		
		IF fbOnTrigger.Q THEN
			Restart := TRUE;
		END_IF

		IF Restart THEN
			Busy := TRUE;

			(* check initialization *)
			IF NOT InitDone AND NOT fbAdsReadModulo.BUSY AND NOT TcMcGlobal.fbADSRDDEVINFO.BUSY THEN
				(* initialization error *)
				Busy := fbAdsReadModulo.BUSY;
				Error := fbAdsReadModulo.ERR;
				ErrorID := fbAdsReadModulo.ERRID;
				fbAdsReadModulo(READ:=FALSE);	(* initialize again during next cycle *)
				Restart := FALSE;	(* error *)
			ELSIF InitDone AND NOT TcMcGlobal.fbADSRDDEVINFO.BUSY THEN;
				(* initialization was okay - check input parameters *)

				IF NOT fbADSwrite.BUSY THEN
					(* initialization *)
					Done := FALSE;
					Error := FALSE;
					ErrorID := 0;
					CommandAborted := FALSE;
					RecordedPosition := 0;
					fbADSwrite(WRITE:=FALSE); (* reset *)
					fbAdsReadValid(READ:=FALSE);
					fbAdsReadValue(READ:=FALSE);
					fbAdsReadState(READ:=FALSE);
					TimerAdsReadState(IN:=FALSE);
					RtrigPlcEvent(CLK:=TriggerInput.PlcEvent);
					FtrigPlcEvent(CLK:=TriggerInput.PlcEvent);
					LastTouchProbeValue := TouchProbeValue;
					LastTouchProbeCounter := TouchProbeCounter;
					Restart := FALSE;
					FOR i := 1 TO 4 DO
						TouchProbeInactiveCounter[i] := 0;
					END_FOR
				END_IF

				IF TriggerInput.Mode = TOUCHPROBEMODE_SINGLE_COMPATIBILITYMODE THEN
					CASE TriggerInput.Edge OF
						RisingEdge :
							IndexOffset := 16#201;
						FallingEdge:
							IndexOffset := 16#202;
					ELSE (* case *)
						Error := TRUE;
						ErrorID := MC_ERROR_INVALID_TOUCH_PROBE;
					END_CASE
				ELSE
					IF TcMcGlobal.NcDeviceInfoNcVersion > 16#020B07DD THEN
						IndexOffset := 16#200;  (* new from 2.11 NC driver 2014 *)
					ELSE
						(* new probe mode with old NC driver not possible *)
						Error := TRUE;
						ErrorID := MC_ERROR_INVALID_TOUCH_PROBE;
					END_IF
				END_IF

				IF TriggerInput.EncoderID > 255 THEN
					Error := TRUE;
					ErrorID := MC_ERROR_INVALID_TOUCH_PROBE;
				END_IF

				IF NOT Error THEN
					CASE TriggerInput.TouchProbe OF
						TouchProbe1,
						TouchProbe2,
						TouchProbe3,
						TouchProbe4:
							(* activate latch *)
							iTriggerInput := TriggerInput; (* save local copy *)
							ActTouchProbeActivate();
							iState := STATE_ORDER;

						PlcEvent:
							(* no action necessary here *);
							TriggerInput.ProbeState := TouchProbeActivated;
							iTriggerInput := TriggerInput; (* save local copy *)
							iState := STATE_WAITING;
					ELSE
						Error := TRUE;
						ErrorID := MC_ERROR_INVALID_TOUCH_PROBE;
					END_CASE
				END_IF
			END_IF
		END_IF

	STATE_ORDER :	(* wait until probe is activated *)
		ActTouchProbeActivate();

	STATE_WAITING : (* wait until touch probe was trigerred *)
		CASE iTriggerInput.TouchProbe OF (* type of touch probe *)
			TouchProbe1,
			TouchProbe2,
			TouchProbe3,
			TouchProbe4:
				IF TcMcGlobal.NcDeviceInfoNcVersion > 16#020B07DD AND stTouchProbeActivation.Mode<>TOUCHPROBEMODE_SINGLE_COMPATIBILITYMODE THEN
					(* new touch probe interface since TwinCAT 2.11 Nc-Driver 2014 *)
					ActTouchProbeMonitoring();
				ELSE
					(* classic touch probe interface until TwinCAT 2.11 Nc-Driver 2013 *)
					ActTouchProbeMonitorLatchValid();
					IF iState=STATE_WAITING THEN (* still not triggered *)
						ActTouchProbeMonitorActivity();
					END_IF
				END_IF

			(* CASE PlcEvent *)
			PlcEvent : (* touch proble will be triggered through a PLC signal (iTriggerInput.PlcEvent) *)
				ActTouchProbeMonitorPlcEvent();
		END_CASE (* type of touch probe *)

		IF NOT Done AND (TriggerInput.ProbeState = TouchProbeAborted) THEN
			(* function block has been aborted by an external MC_AbortTrigger *)
			CommandAborted := TRUE;
			iState := STATE_INITIALIZATION;
		END_IF

		IF TriggerInput.Mode = TOUCHPROBEMODE_CONTINOUS THEN
			(* check if probe triggered, then restart probe *)
			IF Done AND Execute THEN
(*				fbAdsReadState(READ:=FALSE); *)
(*				LastTouchProbeValue := TouchProbeValue;
				LastTouchProbeCounter := TouchProbeCounter;
				fbAdsReadLatchStatus(WRTRD:=TRUE); *)(* retrigger *)
				iState := STATE_WAITING; (* keep on waiting for next trigger *)
			ELSIF NOT Execute THEN (* abort trigger *)
				stTouchProbeDeactivation.TouchProbe := iTriggerInput.TouchProbe;
				stTouchProbeDeactivation.Edge := iTriggerInput.Edge;
				fbADSwrite(	WRITE:=FALSE); (* reset *)
				fbADSwrite(	NETID:= TcMcGlobal.NCNETID_TCMC,
							PORT:=AMSPORT_R0_NCSAF ,
							IDXGRP:=16#5200+TriggerInput.EncoderID ,
							IDXOFFS:=16#205,	(* deactivate touch probe *)
							LEN:= SIZEOF(stTouchProbeDeactivation),
							SRCADDR:=ADR(stTouchProbeDeactivation),
							WRITE:=TRUE ,
							TMOUT:=TcMcGlobal.tADSTimeOut);
				iState := 30000;
			END_IF
		END_IF

		IF iState<> STATE_WAITING THEN
			(* leave the waiting state now *)
			TriggerInput.ProbeState := TouchProbeInactive;
			fbAdsReadModulo(READ:=FALSE);	(* initialize again during next cycle *)
		END_IF

	30000 : (* abort trigger *)
		fbADSwrite();
		IF NOT fbAdsWrite.BUSY THEN
			IF fbAdsWrite.ERR THEN
				Error := fbAdsWrite.ERR;
				ErrorID := fbAdsWrite.ERRID;
			END_IF
			iState := STATE_INITIALIZATION;
		END_IF

END_CASE

ADSbusy := fbAdsWrite.BUSY OR fbAdsReadValid.BUSY OR fbAdsReadValue.BUSY OR fbAdsReadState.BUSY OR fbAdsReadModulo.BUSY;
IF iState=STATE_INITIALIZATION AND NOT Restart THEN
	(* reset Busy immediately  when sequence ends *)
	Busy := FALSE;
END_IF

ACTION ActTouchProbeActivate:
(* start the touch probe sequence *)

(*LatchID := iTriggerInput.TouchProbe;*)
TriggerInput.ProbeState := TouchProbeActivated;
iTriggerInput.ProbeState := TouchProbeActivated;

(* read version of NC *)
(*
IF TcMcGlobal.NcDeviceInfoNcVersion=0 THEN
	TcMcGlobal.ReadDeviceInfo;
END_IF
*)

stTouchProbeActivation.TouchProbe := iTriggerInput.TouchProbe;
stTouchProbeActivation.Edge := iTriggerInput.Edge;
stTouchProbeActivation.Mode := iTriggerInput.Mode;
stTouchProbeActivation.SignalSource := iTriggerInput.SignalSource;	(* 20110218 KSt *)

IF stTouchProbeActivation.Mode = TOUCHPROBEMODE_SINGLE_COMPATIBILITYMODE THEN
	fbADSwrite(	NETID:= TcMcGlobal.NCNETID_TCMC,
				PORT:=AMSPORT_R0_NCSAF ,
				IDXGRP:=16#5200+iTriggerInput.EncoderID ,
				IDXOFFS:=IndexOffset,
				LEN:=0,
				SRCADDR:=ADR(stTouchProbeActivation),
				WRITE:=TRUE ,
				TMOUT:=TcMcGlobal.tADSTimeOut);
ELSE
	fbADSwrite(	NETID:= TcMcGlobal.NCNETID_TCMC,
				PORT:=AMSPORT_R0_NCSAF ,
				IDXGRP:=16#5200+iTriggerInput.EncoderID ,
				IDXOFFS:=IndexOffset,
				LEN:=SIZEOF(stTouchProbeActivation),
				SRCADDR:=ADR(stTouchProbeActivation),
				WRITE:=TRUE ,
				TMOUT:=TcMcGlobal.tADSTimeOut);
END_IF

IF NOT fbADSwrite.BUSY THEN
	IF fbADSwrite.ERR THEN
		Error := fbADSwrite.ERR;
		ErrorID := fbADSwrite.ERRID;
	END_IF
	IF NOT Error AND iTriggerInput.ProbeState = TouchProbeAborted THEN
		(* Synchronization error between MC_TouchProbe and MC_AbortTrigger *)
		Error := TRUE;
		ErrorID := MC_ERROR_TOUCH_PROBE_DEACTIVATED;
	END_IF
	iTriggerInput.ProbeState := SEL( Error, TouchProbeActivated, TouchProbeInactive );
	iState := SEL( Error, STATE_WAITING, STATE_INITIALIZATION);
END_IF
END_ACTION

ACTION ActTouchProbeMonitorActivity:
(* check if latch is still active *)
TimerAdsReadState(IN := NOT TimerAdsReadState.q , PT:=T#1s);
IF TimerAdsReadState.q OR fbAdsReadState.BUSY THEN
	fbAdsReadState(	NETID:= TcMcGlobal.NCNETID_TCMC,
				PORT:=AMSPORT_R0_NCSAF ,
				IDXGRP:=16#5100+TriggerInput.EncoderID ,
				IDXOFFS:= 16#201,
				LEN:= SIZEOF(TouchProbeActive[1]),
				DESTADDR:=ADR(TouchProbeActive) ,
				READ:=TRUE ,
				TMOUT:=TcMcGlobal.tADSTimeOut );
	IF NOT fbAdsReadState.BUSY THEN
		IF fbAdsReadState.ERR THEN
			Error := TRUE;
			ErrorID := fbAdsReadState.ERRID;
		ELSE
			IF TouchProbeActive[TriggerInput.TouchProbe]<>1 THEN
				TouchProbeInactiveCounter[TriggerInput.TouchProbe] := TouchProbeInactiveCounter[TriggerInput.TouchProbe] + 1;
				IF TouchProbeInactiveCounter[TriggerInput.TouchProbe] > 1 THEN
					(* error condition when the probing sequence is inactive more than once *)
					Error := TRUE;
					ErrorID := MC_ERROR_TOUCH_PROBE_DEACTIVATED;
					CommandAborted := TRUE;
					iState := STATE_INITIALIZATION;
				END_IF
			END_IF
		END_IF
		fbAdsReadState(READ:=FALSE); (* reset *)
	END_IF
END_IF
END_ACTION

ACTION ActTouchProbeMonitoring:

(* 	monitor if the touch probe has been triggered and if it is still active *)

(* 	new touch probe interface since 4/2010
	This action is only used with the new interface 
*)

Done := FALSE;		(* default *)
RecordedPosition := 0;	(* default *)

(* check if latch is still active and check for valid latch *)
TimerAdsReadState(IN := NOT TimerAdsReadState.q , PT:=T#1s);
IF ExternalLatchValid OR TimerAdsReadState.q OR fbAdsReadLatchStatus.BUSY THEN
	(* request for this probe unit *)
	stTouchProbeStatusRequest.TouchProbe := iTriggerInput.TouchProbe;

	fbAdsReadLatchStatus(
		NETID:= TcMcGlobal.NCNETID_TCMC,
		PORT:=AMSPORT_R0_NCSAF ,
		IDXGRP:=16#5100+iTriggerInput.EncoderID ,
		IDXOFFS:= 16#200,
		WRITELEN:= SIZEOF(stTouchProbeStatusRequest),
		READLEN:= SIZEOF(stTouchProbeStatusResponse),
		SRCADDR:= ADR(stTouchProbeStatusRequest),
		DESTADDR:= ADR(stTouchProbeStatusResponse),
		WRTRD:= TRUE,
		TMOUT:= TcMcGlobal.tADSTimeOut );

